DATA_BLOCK "Parameter"
{ S7_Optimized_Access := 'TRUE' }
VERSION : 0.1
NON_RETAIN
// ATTRIBUTES
// AUTO_NUMBER = False
// BLOCK_NUMBER = 170
// END_ATTRIBUTES
   VAR RETAIN
      AxisRun : Struct
         Axis { S7_SetPoint := 'False'} : Array[1..15] of "ServoType_UDT";
      END_STRUCT;
      AxisNuw : Struct
         Axis { S7_SetPoint := 'False'} : Array[1..15] of "ServoType_UDT";
      END_STRUCT;
      AxisDisplay : Struct
         Axis { S7_SetPoint := 'False'} : Array[1..15] of "ServoType_UDT";
      END_STRUCT;
      AxisSave : Struct
         Axis { S7_SetPoint := 'False'} : Array[1..15] of "ServoType_UDT";
      END_STRUCT;
      AxisStore : Array[1..15] of Struct
         Axis { S7_SetPoint := 'False'} : Array[1..15] of "ServoType_UDT";
      END_STRUCT;
   END_VAR


BEGIN
   AxisRun.Axis[1].Pos1.Position := 3.419;
   AxisRun.Axis[1].Pos1.Speed := 10000;
   AxisRun.Axis[1].Pos1.Reached := FALSE;
   AxisRun.Axis[1].Pos2.Position := 48.386;
   AxisRun.Axis[1].Pos2.Speed := 10000;
   AxisRun.Axis[1].Pos2.Reached := FALSE;
   AxisRun.Axis[1].Pos3.Position := 93.294;
   AxisRun.Axis[1].Pos3.Speed := 10000;
   AxisRun.Axis[1].Pos3.Reached := FALSE;
   AxisRun.Axis[1].Pos4.Position := 138.335;
   AxisRun.Axis[1].Pos4.Speed := 10000;
   AxisRun.Axis[1].Pos4.Reached := FALSE;
   AxisRun.Axis[1].Pos5.Position := 183.464;
   AxisRun.Axis[1].Pos5.Speed := 10000;
   AxisRun.Axis[1].Pos5.Reached := FALSE;
   AxisRun.Axis[1].Pos6.Position := 228.443;
   AxisRun.Axis[1].Pos6.Speed := 10000;
   AxisRun.Axis[1].Pos6.Reached := FALSE;
   AxisRun.Axis[1].Pos7.Position := 273.535;
   AxisRun.Axis[1].Pos7.Speed := 10000;
   AxisRun.Axis[1].Pos7.Reached := FALSE;
   AxisRun.Axis[1].Pos8.Position := 318.25;
   AxisRun.Axis[1].Pos8.Speed := 10000;
   AxisRun.Axis[1].Pos8.Reached := FALSE;
   AxisRun.Axis[1].Pos9.Position := 0.0;
   AxisRun.Axis[1].Pos9.Speed := 0;
   AxisRun.Axis[1].Pos9.Reached := FALSE;
   AxisRun.Axis[1].Pos10.Position := 0.0;
   AxisRun.Axis[1].Pos10.Speed := 0;
   AxisRun.Axis[1].Pos10.Reached := FALSE;
   AxisRun.Axis[1].Pos11.Position := 0.0;
   AxisRun.Axis[1].Pos11.Speed := 0;
   AxisRun.Axis[1].Pos11.Reached := FALSE;
   AxisRun.Axis[1].Pos12.Position := 0.0;
   AxisRun.Axis[1].Pos12.Speed := 0;
   AxisRun.Axis[1].Pos12.Reached := FALSE;
   AxisRun.Axis[1].Pos13.Position := 0.0;
   AxisRun.Axis[1].Pos13.Speed := 0;
   AxisRun.Axis[1].Pos13.Reached := FALSE;
   AxisRun.Axis[1].Pos14.Position := 0.0;
   AxisRun.Axis[1].Pos14.Speed := 0;
   AxisRun.Axis[1].Pos14.Reached := FALSE;
   AxisRun.Axis[1].Pos15.Position := 0.0;
   AxisRun.Axis[1].Pos15.Speed := 0;
   AxisRun.Axis[1].Pos15.Reached := FALSE;
   AxisRun.Axis[1].Pos16.Position := 0.0;
   AxisRun.Axis[1].Pos16.Speed := 0;
   AxisRun.Axis[1].Pos16.Reached := FALSE;
   AxisRun.Axis[1].Pos17.Position := 0.0;
   AxisRun.Axis[1].Pos17.Speed := 0;
   AxisRun.Axis[1].Pos17.Reached := FALSE;
   AxisRun.Axis[1].Pos18.Position := 0.0;
   AxisRun.Axis[1].Pos18.Speed := 0;
   AxisRun.Axis[1].Pos18.Reached := FALSE;
   AxisRun.Axis[1].Pos19.Position := 0.0;
   AxisRun.Axis[1].Pos19.Speed := 0;
   AxisRun.Axis[1].Pos19.Reached := FALSE;
   AxisRun.Axis[1].Pos20.Position := 0.0;
   AxisRun.Axis[1].Pos20.Speed := 0;
   AxisRun.Axis[1].Pos20.Reached := FALSE;
   AxisRun.Axis[1].Pos21.Position := 0.0;
   AxisRun.Axis[1].Pos21.Speed := 0;
   AxisRun.Axis[1].Pos21.Reached := FALSE;
   AxisRun.Axis[1].Pos22.Position := 0.0;
   AxisRun.Axis[1].Pos22.Speed := 0;
   AxisRun.Axis[1].Pos22.Reached := FALSE;
   AxisRun.Axis[1].Pos23.Position := 0.0;
   AxisRun.Axis[1].Pos23.Speed := 0;
   AxisRun.Axis[1].Pos23.Reached := FALSE;
   AxisRun.Axis[1].Pos24.Position := 0.0;
   AxisRun.Axis[1].Pos24.Speed := 0;
   AxisRun.Axis[1].Pos24.Reached := FALSE;
   AxisRun.Axis[1].Pos25.Position := 0.0;
   AxisRun.Axis[1].Pos25.Speed := 0;
   AxisRun.Axis[1].Pos25.Reached := FALSE;
   AxisRun.Axis[1].Pos26.Position := 0.0;
   AxisRun.Axis[1].Pos26.Speed := 0;
   AxisRun.Axis[1].Pos26.Reached := FALSE;
   AxisRun.Axis[1].Pos27.Position := 0.0;
   AxisRun.Axis[1].Pos27.Speed := 0;
   AxisRun.Axis[1].Pos27.Reached := FALSE;
   AxisRun.Axis[1].Pos28.Position := 0.0;
   AxisRun.Axis[1].Pos28.Speed := 0;
   AxisRun.Axis[1].Pos28.Reached := FALSE;
   AxisRun.Axis[1].Pos29.Position := 0.0;
   AxisRun.Axis[1].Pos29.Speed := 0;
   AxisRun.Axis[1].Pos29.Reached := FALSE;
   AxisRun.Axis[1].Pos30.Position := 0.0;
   AxisRun.Axis[1].Pos30.Speed := 0;
   AxisRun.Axis[1].Pos30.Reached := FALSE;
   AxisRun.Axis[2].Pos1.Position := 0.0;
   AxisRun.Axis[2].Pos1.Speed := 10000;
   AxisRun.Axis[2].Pos1.Reached := FALSE;
   AxisRun.Axis[2].Pos2.Position := 450.0;
   AxisRun.Axis[2].Pos2.Speed := 10000;
   AxisRun.Axis[2].Pos2.Reached := FALSE;
   AxisRun.Axis[2].Pos3.Position := 900.0;
   AxisRun.Axis[2].Pos3.Speed := 10000;
   AxisRun.Axis[2].Pos3.Reached := FALSE;
   AxisRun.Axis[2].Pos4.Position := 135.0;
   AxisRun.Axis[2].Pos4.Speed := 10000;
   AxisRun.Axis[2].Pos4.Reached := FALSE;
   AxisRun.Axis[2].Pos5.Position := 180.0;
   AxisRun.Axis[2].Pos5.Speed := 10000;
   AxisRun.Axis[2].Pos5.Reached := FALSE;
   AxisRun.Axis[2].Pos6.Position := 225.0;
   AxisRun.Axis[2].Pos6.Speed := 10000;
   AxisRun.Axis[2].Pos6.Reached := FALSE;
   AxisRun.Axis[2].Pos7.Position := 270.0;
   AxisRun.Axis[2].Pos7.Speed := 10000;
   AxisRun.Axis[2].Pos7.Reached := FALSE;
   AxisRun.Axis[2].Pos8.Position := 315.0;
   AxisRun.Axis[2].Pos8.Speed := 10000;
   AxisRun.Axis[2].Pos8.Reached := FALSE;
   AxisRun.Axis[2].Pos9.Position := 0.0;
   AxisRun.Axis[2].Pos9.Speed := 0;
   AxisRun.Axis[2].Pos9.Reached := FALSE;
   AxisRun.Axis[2].Pos10.Position := 0.0;
   AxisRun.Axis[2].Pos10.Speed := 0;
   AxisRun.Axis[2].Pos10.Reached := FALSE;
   AxisRun.Axis[2].Pos11.Position := 0.0;
   AxisRun.Axis[2].Pos11.Speed := 0;
   AxisRun.Axis[2].Pos11.Reached := FALSE;
   AxisRun.Axis[2].Pos12.Position := 0.0;
   AxisRun.Axis[2].Pos12.Speed := 0;
   AxisRun.Axis[2].Pos12.Reached := FALSE;
   AxisRun.Axis[2].Pos13.Position := 0.0;
   AxisRun.Axis[2].Pos13.Speed := 0;
   AxisRun.Axis[2].Pos13.Reached := FALSE;
   AxisRun.Axis[2].Pos14.Position := 0.0;
   AxisRun.Axis[2].Pos14.Speed := 0;
   AxisRun.Axis[2].Pos14.Reached := FALSE;
   AxisRun.Axis[2].Pos15.Position := 0.0;
   AxisRun.Axis[2].Pos15.Speed := 0;
   AxisRun.Axis[2].Pos15.Reached := FALSE;
   AxisRun.Axis[2].Pos16.Position := 0.0;
   AxisRun.Axis[2].Pos16.Speed := 0;
   AxisRun.Axis[2].Pos16.Reached := FALSE;
   AxisRun.Axis[2].Pos17.Position := 0.0;
   AxisRun.Axis[2].Pos17.Speed := 0;
   AxisRun.Axis[2].Pos17.Reached := FALSE;
   AxisRun.Axis[2].Pos18.Position := 0.0;
   AxisRun.Axis[2].Pos18.Speed := 0;
   AxisRun.Axis[2].Pos18.Reached := FALSE;
   AxisRun.Axis[2].Pos19.Position := 0.0;
   AxisRun.Axis[2].Pos19.Speed := 0;
   AxisRun.Axis[2].Pos19.Reached := FALSE;
   AxisRun.Axis[2].Pos20.Position := 0.0;
   AxisRun.Axis[2].Pos20.Speed := 0;
   AxisRun.Axis[2].Pos20.Reached := FALSE;
   AxisRun.Axis[2].Pos21.Position := 0.0;
   AxisRun.Axis[2].Pos21.Speed := 0;
   AxisRun.Axis[2].Pos21.Reached := FALSE;
   AxisRun.Axis[2].Pos22.Position := 0.0;
   AxisRun.Axis[2].Pos22.Speed := 0;
   AxisRun.Axis[2].Pos22.Reached := FALSE;
   AxisRun.Axis[2].Pos23.Position := 0.0;
   AxisRun.Axis[2].Pos23.Speed := 0;
   AxisRun.Axis[2].Pos23.Reached := FALSE;
   AxisRun.Axis[2].Pos24.Position := 0.0;
   AxisRun.Axis[2].Pos24.Speed := 0;
   AxisRun.Axis[2].Pos24.Reached := FALSE;
   AxisRun.Axis[2].Pos25.Position := 0.0;
   AxisRun.Axis[2].Pos25.Speed := 0;
   AxisRun.Axis[2].Pos25.Reached := FALSE;
   AxisRun.Axis[2].Pos26.Position := 0.0;
   AxisRun.Axis[2].Pos26.Speed := 0;
   AxisRun.Axis[2].Pos26.Reached := FALSE;
   AxisRun.Axis[2].Pos27.Position := 0.0;
   AxisRun.Axis[2].Pos27.Speed := 0;
   AxisRun.Axis[2].Pos27.Reached := FALSE;
   AxisRun.Axis[2].Pos28.Position := 0.0;
   AxisRun.Axis[2].Pos28.Speed := 0;
   AxisRun.Axis[2].Pos28.Reached := FALSE;
   AxisRun.Axis[2].Pos29.Position := 0.0;
   AxisRun.Axis[2].Pos29.Speed := 0;
   AxisRun.Axis[2].Pos29.Reached := FALSE;
   AxisRun.Axis[2].Pos30.Position := 0.0;
   AxisRun.Axis[2].Pos30.Speed := 0;
   AxisRun.Axis[2].Pos30.Reached := FALSE;
   AxisRun.Axis[3].Pos1.Position := 0.0;
   AxisRun.Axis[3].Pos1.Speed := 20000;
   AxisRun.Axis[3].Pos1.Reached := FALSE;
   AxisRun.Axis[3].Pos2.Position := 490.0;
   AxisRun.Axis[3].Pos2.Speed := 10000;
   AxisRun.Axis[3].Pos2.Reached := FALSE;
   AxisRun.Axis[3].Pos3.Position := 490.0;
   AxisRun.Axis[3].Pos3.Speed := 10000;
   AxisRun.Axis[3].Pos3.Reached := FALSE;
   AxisRun.Axis[3].Pos4.Position := 490.0;
   AxisRun.Axis[3].Pos4.Speed := 10000;
   AxisRun.Axis[3].Pos4.Reached := FALSE;
   AxisRun.Axis[3].Pos5.Position := 0.0;
   AxisRun.Axis[3].Pos5.Speed := 0;
   AxisRun.Axis[3].Pos5.Reached := FALSE;
   AxisRun.Axis[3].Pos6.Position := 490.0;
   AxisRun.Axis[3].Pos6.Speed := 10000;
   AxisRun.Axis[3].Pos6.Reached := FALSE;
   AxisRun.Axis[3].Pos7.Position := 90.0;
   AxisRun.Axis[3].Pos7.Speed := 10000;
   AxisRun.Axis[3].Pos7.Reached := FALSE;
   AxisRun.Axis[3].Pos8.Position := 180.0;
   AxisRun.Axis[3].Pos8.Speed := 10000;
   AxisRun.Axis[3].Pos8.Reached := FALSE;
   AxisRun.Axis[3].Pos9.Position := 270.0;
   AxisRun.Axis[3].Pos9.Speed := 10000;
   AxisRun.Axis[3].Pos9.Reached := FALSE;
   AxisRun.Axis[3].Pos10.Position := 0.0;
   AxisRun.Axis[3].Pos10.Speed := 0;
   AxisRun.Axis[3].Pos10.Reached := FALSE;
   AxisRun.Axis[3].Pos11.Position := 0.0;
   AxisRun.Axis[3].Pos11.Speed := 0;
   AxisRun.Axis[3].Pos11.Reached := FALSE;
   AxisRun.Axis[3].Pos12.Position := 0.0;
   AxisRun.Axis[3].Pos12.Speed := 0;
   AxisRun.Axis[3].Pos12.Reached := FALSE;
   AxisRun.Axis[3].Pos13.Position := 0.0;
   AxisRun.Axis[3].Pos13.Speed := 0;
   AxisRun.Axis[3].Pos13.Reached := FALSE;
   AxisRun.Axis[3].Pos14.Position := 0.0;
   AxisRun.Axis[3].Pos14.Speed := 0;
   AxisRun.Axis[3].Pos14.Reached := FALSE;
   AxisRun.Axis[3].Pos15.Position := 0.0;
   AxisRun.Axis[3].Pos15.Speed := 0;
   AxisRun.Axis[3].Pos15.Reached := FALSE;
   AxisRun.Axis[3].Pos16.Position := 0.0;
   AxisRun.Axis[3].Pos16.Speed := 0;
   AxisRun.Axis[3].Pos16.Reached := FALSE;
   AxisRun.Axis[3].Pos17.Position := 0.0;
   AxisRun.Axis[3].Pos17.Speed := 0;
   AxisRun.Axis[3].Pos17.Reached := FALSE;
   AxisRun.Axis[3].Pos18.Position := 0.0;
   AxisRun.Axis[3].Pos18.Speed := 0;
   AxisRun.Axis[3].Pos18.Reached := FALSE;
   AxisRun.Axis[3].Pos19.Position := 0.0;
   AxisRun.Axis[3].Pos19.Speed := 0;
   AxisRun.Axis[3].Pos19.Reached := FALSE;
   AxisRun.Axis[3].Pos20.Position := 0.0;
   AxisRun.Axis[3].Pos20.Speed := 0;
   AxisRun.Axis[3].Pos20.Reached := FALSE;
   AxisRun.Axis[3].Pos21.Position := 0.0;
   AxisRun.Axis[3].Pos21.Speed := 0;
   AxisRun.Axis[3].Pos21.Reached := FALSE;
   AxisRun.Axis[3].Pos22.Position := 0.0;
   AxisRun.Axis[3].Pos22.Speed := 0;
   AxisRun.Axis[3].Pos22.Reached := FALSE;
   AxisRun.Axis[3].Pos23.Position := 0.0;
   AxisRun.Axis[3].Pos23.Speed := 0;
   AxisRun.Axis[3].Pos23.Reached := FALSE;
   AxisRun.Axis[3].Pos24.Position := 0.0;
   AxisRun.Axis[3].Pos24.Speed := 0;
   AxisRun.Axis[3].Pos24.Reached := FALSE;
   AxisRun.Axis[3].Pos25.Position := 0.0;
   AxisRun.Axis[3].Pos25.Speed := 0;
   AxisRun.Axis[3].Pos25.Reached := FALSE;
   AxisRun.Axis[3].Pos26.Position := 0.0;
   AxisRun.Axis[3].Pos26.Speed := 0;
   AxisRun.Axis[3].Pos26.Reached := FALSE;
   AxisRun.Axis[3].Pos27.Position := 0.0;
   AxisRun.Axis[3].Pos27.Speed := 0;
   AxisRun.Axis[3].Pos27.Reached := FALSE;
   AxisRun.Axis[3].Pos28.Position := 0.0;
   AxisRun.Axis[3].Pos28.Speed := 0;
   AxisRun.Axis[3].Pos28.Reached := FALSE;
   AxisRun.Axis[3].Pos29.Position := 0.0;
   AxisRun.Axis[3].Pos29.Speed := 0;
   AxisRun.Axis[3].Pos29.Reached := FALSE;
   AxisRun.Axis[3].Pos30.Position := 0.0;
   AxisRun.Axis[3].Pos30.Speed := 0;
   AxisRun.Axis[3].Pos30.Reached := FALSE;
   AxisRun.Axis[4].Pos1.Position := 3.585;
   AxisRun.Axis[4].Pos1.Speed := 10000;
   AxisRun.Axis[4].Pos1.Reached := FALSE;
   AxisRun.Axis[4].Pos2.Position := 48.61;
   AxisRun.Axis[4].Pos2.Speed := 10000;
   AxisRun.Axis[4].Pos2.Reached := FALSE;
   AxisRun.Axis[4].Pos3.Position := 93.637;
   AxisRun.Axis[4].Pos3.Speed := 10000;
   AxisRun.Axis[4].Pos3.Reached := FALSE;
   AxisRun.Axis[4].Pos4.Position := 138.606;
   AxisRun.Axis[4].Pos4.Speed := 10000;
   AxisRun.Axis[4].Pos4.Reached := FALSE;
   AxisRun.Axis[4].Pos5.Position := 183.388;
   AxisRun.Axis[4].Pos5.Speed := 10000;
   AxisRun.Axis[4].Pos5.Reached := FALSE;
   AxisRun.Axis[4].Pos6.Position := 228.458;
   AxisRun.Axis[4].Pos6.Speed := 10000;
   AxisRun.Axis[4].Pos6.Reached := FALSE;
   AxisRun.Axis[4].Pos7.Position := 273.513;
   AxisRun.Axis[4].Pos7.Speed := 10000;
   AxisRun.Axis[4].Pos7.Reached := FALSE;
   AxisRun.Axis[4].Pos8.Position := 318.501;
   AxisRun.Axis[4].Pos8.Speed := 10000;
   AxisRun.Axis[4].Pos8.Reached := FALSE;
   AxisRun.Axis[4].Pos9.Position := 0.0;
   AxisRun.Axis[4].Pos9.Speed := 0;
   AxisRun.Axis[4].Pos9.Reached := FALSE;
   AxisRun.Axis[4].Pos10.Position := 0.0;
   AxisRun.Axis[4].Pos10.Speed := 0;
   AxisRun.Axis[4].Pos10.Reached := FALSE;
   AxisRun.Axis[4].Pos11.Position := 0.0;
   AxisRun.Axis[4].Pos11.Speed := 0;
   AxisRun.Axis[4].Pos11.Reached := FALSE;
   AxisRun.Axis[4].Pos12.Position := 0.0;
   AxisRun.Axis[4].Pos12.Speed := 0;
   AxisRun.Axis[4].Pos12.Reached := FALSE;
   AxisRun.Axis[4].Pos13.Position := 0.0;
   AxisRun.Axis[4].Pos13.Speed := 0;
   AxisRun.Axis[4].Pos13.Reached := FALSE;
   AxisRun.Axis[4].Pos14.Position := 0.0;
   AxisRun.Axis[4].Pos14.Speed := 0;
   AxisRun.Axis[4].Pos14.Reached := FALSE;
   AxisRun.Axis[4].Pos15.Position := 0.0;
   AxisRun.Axis[4].Pos15.Speed := 0;
   AxisRun.Axis[4].Pos15.Reached := FALSE;
   AxisRun.Axis[4].Pos16.Position := 0.0;
   AxisRun.Axis[4].Pos16.Speed := 0;
   AxisRun.Axis[4].Pos16.Reached := FALSE;
   AxisRun.Axis[4].Pos17.Position := 0.0;
   AxisRun.Axis[4].Pos17.Speed := 0;
   AxisRun.Axis[4].Pos17.Reached := FALSE;
   AxisRun.Axis[4].Pos18.Position := 0.0;
   AxisRun.Axis[4].Pos18.Speed := 0;
   AxisRun.Axis[4].Pos18.Reached := FALSE;
   AxisRun.Axis[4].Pos19.Position := 0.0;
   AxisRun.Axis[4].Pos19.Speed := 0;
   AxisRun.Axis[4].Pos19.Reached := FALSE;
   AxisRun.Axis[4].Pos20.Position := 0.0;
   AxisRun.Axis[4].Pos20.Speed := 0;
   AxisRun.Axis[4].Pos20.Reached := FALSE;
   AxisRun.Axis[4].Pos21.Position := 0.0;
   AxisRun.Axis[4].Pos21.Speed := 0;
   AxisRun.Axis[4].Pos21.Reached := FALSE;
   AxisRun.Axis[4].Pos22.Position := 0.0;
   AxisRun.Axis[4].Pos22.Speed := 0;
   AxisRun.Axis[4].Pos22.Reached := FALSE;
   AxisRun.Axis[4].Pos23.Position := 0.0;
   AxisRun.Axis[4].Pos23.Speed := 0;
   AxisRun.Axis[4].Pos23.Reached := FALSE;
   AxisRun.Axis[4].Pos24.Position := 0.0;
   AxisRun.Axis[4].Pos24.Speed := 0;
   AxisRun.Axis[4].Pos24.Reached := FALSE;
   AxisRun.Axis[4].Pos25.Position := 0.0;
   AxisRun.Axis[4].Pos25.Speed := 0;
   AxisRun.Axis[4].Pos25.Reached := FALSE;
   AxisRun.Axis[4].Pos26.Position := 0.0;
   AxisRun.Axis[4].Pos26.Speed := 0;
   AxisRun.Axis[4].Pos26.Reached := FALSE;
   AxisRun.Axis[4].Pos27.Position := 0.0;
   AxisRun.Axis[4].Pos27.Speed := 0;
   AxisRun.Axis[4].Pos27.Reached := FALSE;
   AxisRun.Axis[4].Pos28.Position := 0.0;
   AxisRun.Axis[4].Pos28.Speed := 0;
   AxisRun.Axis[4].Pos28.Reached := FALSE;
   AxisRun.Axis[4].Pos29.Position := 0.0;
   AxisRun.Axis[4].Pos29.Speed := 0;
   AxisRun.Axis[4].Pos29.Reached := FALSE;
   AxisRun.Axis[4].Pos30.Position := 0.0;
   AxisRun.Axis[4].Pos30.Speed := 0;
   AxisRun.Axis[4].Pos30.Reached := FALSE;
   AxisRun.Axis[5].Pos1.Position := 143.76;
   AxisRun.Axis[5].Pos1.Speed := 200;
   AxisRun.Axis[5].Pos1.Reached := FALSE;
   AxisRun.Axis[5].Pos2.Position := 143.76;
   AxisRun.Axis[5].Pos2.Speed := 200;
   AxisRun.Axis[5].Pos2.Reached := FALSE;
   AxisRun.Axis[5].Pos3.Position := 137.76;
   AxisRun.Axis[5].Pos3.Speed := 200;
   AxisRun.Axis[5].Pos3.Reached := FALSE;
   AxisRun.Axis[5].Pos4.Position := 130.36;
   AxisRun.Axis[5].Pos4.Speed := 200;
   AxisRun.Axis[5].Pos4.Reached := FALSE;
   AxisRun.Axis[5].Pos5.Position := 124.16;
   AxisRun.Axis[5].Pos5.Speed := 200;
   AxisRun.Axis[5].Pos5.Reached := FALSE;
   AxisRun.Axis[5].Pos6.Position := 125.65;
   AxisRun.Axis[5].Pos6.Speed := 200;
   AxisRun.Axis[5].Pos6.Reached := FALSE;
   AxisRun.Axis[5].Pos7.Position := 48.11;
   AxisRun.Axis[5].Pos7.Speed := 200;
   AxisRun.Axis[5].Pos7.Reached := FALSE;
   AxisRun.Axis[5].Pos8.Position := 0.0;
   AxisRun.Axis[5].Pos8.Speed := 200;
   AxisRun.Axis[5].Pos8.Reached := FALSE;
   AxisRun.Axis[5].Pos9.Position := 48.11;
   AxisRun.Axis[5].Pos9.Speed := 200;
   AxisRun.Axis[5].Pos9.Reached := FALSE;
   AxisRun.Axis[5].Pos10.Position := 0.0;
   AxisRun.Axis[5].Pos10.Speed := 0;
   AxisRun.Axis[5].Pos10.Reached := FALSE;
   AxisRun.Axis[5].Pos11.Position := 0.0;
   AxisRun.Axis[5].Pos11.Speed := 0;
   AxisRun.Axis[5].Pos11.Reached := FALSE;
   AxisRun.Axis[5].Pos12.Position := 0.0;
   AxisRun.Axis[5].Pos12.Speed := 0;
   AxisRun.Axis[5].Pos12.Reached := FALSE;
   AxisRun.Axis[5].Pos13.Position := 0.0;
   AxisRun.Axis[5].Pos13.Speed := 0;
   AxisRun.Axis[5].Pos13.Reached := FALSE;
   AxisRun.Axis[5].Pos14.Position := 0.0;
   AxisRun.Axis[5].Pos14.Speed := 0;
   AxisRun.Axis[5].Pos14.Reached := FALSE;
   AxisRun.Axis[5].Pos15.Position := 0.0;
   AxisRun.Axis[5].Pos15.Speed := 0;
   AxisRun.Axis[5].Pos15.Reached := FALSE;
   AxisRun.Axis[5].Pos16.Position := 0.0;
   AxisRun.Axis[5].Pos16.Speed := 0;
   AxisRun.Axis[5].Pos16.Reached := FALSE;
   AxisRun.Axis[5].Pos17.Position := 0.0;
   AxisRun.Axis[5].Pos17.Speed := 0;
   AxisRun.Axis[5].Pos17.Reached := FALSE;
   AxisRun.Axis[5].Pos18.Position := 0.0;
   AxisRun.Axis[5].Pos18.Speed := 0;
   AxisRun.Axis[5].Pos18.Reached := FALSE;
   AxisRun.Axis[5].Pos19.Position := 0.0;
   AxisRun.Axis[5].Pos19.Speed := 0;
   AxisRun.Axis[5].Pos19.Reached := FALSE;
   AxisRun.Axis[5].Pos20.Position := 0.0;
   AxisRun.Axis[5].Pos20.Speed := 0;
   AxisRun.Axis[5].Pos20.Reached := FALSE;
   AxisRun.Axis[5].Pos21.Position := 0.0;
   AxisRun.Axis[5].Pos21.Speed := 0;
   AxisRun.Axis[5].Pos21.Reached := FALSE;
   AxisRun.Axis[5].Pos22.Position := 0.0;
   AxisRun.Axis[5].Pos22.Speed := 0;
   AxisRun.Axis[5].Pos22.Reached := FALSE;
   AxisRun.Axis[5].Pos23.Position := 0.0;
   AxisRun.Axis[5].Pos23.Speed := 0;
   AxisRun.Axis[5].Pos23.Reached := FALSE;
   AxisRun.Axis[5].Pos24.Position := 0.0;
   AxisRun.Axis[5].Pos24.Speed := 0;
   AxisRun.Axis[5].Pos24.Reached := FALSE;
   AxisRun.Axis[5].Pos25.Position := 0.0;
   AxisRun.Axis[5].Pos25.Speed := 0;
   AxisRun.Axis[5].Pos25.Reached := FALSE;
   AxisRun.Axis[5].Pos26.Position := 0.0;
   AxisRun.Axis[5].Pos26.Speed := 0;
   AxisRun.Axis[5].Pos26.Reached := FALSE;
   AxisRun.Axis[5].Pos27.Position := 0.0;
   AxisRun.Axis[5].Pos27.Speed := 0;
   AxisRun.Axis[5].Pos27.Reached := FALSE;
   AxisRun.Axis[5].Pos28.Position := 0.0;
   AxisRun.Axis[5].Pos28.Speed := 0;
   AxisRun.Axis[5].Pos28.Reached := FALSE;
   AxisRun.Axis[5].Pos29.Position := 0.0;
   AxisRun.Axis[5].Pos29.Speed := 0;
   AxisRun.Axis[5].Pos29.Reached := FALSE;
   AxisRun.Axis[5].Pos30.Position := 0.0;
   AxisRun.Axis[5].Pos30.Speed := 0;
   AxisRun.Axis[5].Pos30.Reached := FALSE;
   AxisRun.Axis[6].Pos1.Position := 2.34;
   AxisRun.Axis[6].Pos1.Speed := 200;
   AxisRun.Axis[6].Pos1.Reached := FALSE;
   AxisRun.Axis[6].Pos2.Position := 76.0;
   AxisRun.Axis[6].Pos2.Speed := 200;
   AxisRun.Axis[6].Pos2.Reached := FALSE;
   AxisRun.Axis[6].Pos3.Position := 84.69;
   AxisRun.Axis[6].Pos3.Speed := 200;
   AxisRun.Axis[6].Pos3.Reached := FALSE;
   AxisRun.Axis[6].Pos4.Position := 84.69;
   AxisRun.Axis[6].Pos4.Speed := 200;
   AxisRun.Axis[6].Pos4.Reached := FALSE;
   AxisRun.Axis[6].Pos5.Position := 84.69;
   AxisRun.Axis[6].Pos5.Speed := 200;
   AxisRun.Axis[6].Pos5.Reached := FALSE;
   AxisRun.Axis[6].Pos6.Position := 84.69;
   AxisRun.Axis[6].Pos6.Speed := 200;
   AxisRun.Axis[6].Pos6.Reached := FALSE;
   AxisRun.Axis[6].Pos7.Position := 85.0;
   AxisRun.Axis[6].Pos7.Speed := 200;
   AxisRun.Axis[6].Pos7.Reached := FALSE;
   AxisRun.Axis[6].Pos8.Position := 88.53;
   AxisRun.Axis[6].Pos8.Speed := 200;
   AxisRun.Axis[6].Pos8.Reached := FALSE;
   AxisRun.Axis[6].Pos9.Position := 0.0;
   AxisRun.Axis[6].Pos9.Speed := 0;
   AxisRun.Axis[6].Pos9.Reached := FALSE;
   AxisRun.Axis[6].Pos10.Position := 0.0;
   AxisRun.Axis[6].Pos10.Speed := 0;
   AxisRun.Axis[6].Pos10.Reached := FALSE;
   AxisRun.Axis[6].Pos11.Position := 0.0;
   AxisRun.Axis[6].Pos11.Speed := 0;
   AxisRun.Axis[6].Pos11.Reached := FALSE;
   AxisRun.Axis[6].Pos12.Position := 0.0;
   AxisRun.Axis[6].Pos12.Speed := 0;
   AxisRun.Axis[6].Pos12.Reached := FALSE;
   AxisRun.Axis[6].Pos13.Position := 0.0;
   AxisRun.Axis[6].Pos13.Speed := 0;
   AxisRun.Axis[6].Pos13.Reached := FALSE;
   AxisRun.Axis[6].Pos14.Position := 0.0;
   AxisRun.Axis[6].Pos14.Speed := 0;
   AxisRun.Axis[6].Pos14.Reached := FALSE;
   AxisRun.Axis[6].Pos15.Position := 0.0;
   AxisRun.Axis[6].Pos15.Speed := 0;
   AxisRun.Axis[6].Pos15.Reached := FALSE;
   AxisRun.Axis[6].Pos16.Position := 0.0;
   AxisRun.Axis[6].Pos16.Speed := 0;
   AxisRun.Axis[6].Pos16.Reached := FALSE;
   AxisRun.Axis[6].Pos17.Position := 0.0;
   AxisRun.Axis[6].Pos17.Speed := 0;
   AxisRun.Axis[6].Pos17.Reached := FALSE;
   AxisRun.Axis[6].Pos18.Position := 0.0;
   AxisRun.Axis[6].Pos18.Speed := 0;
   AxisRun.Axis[6].Pos18.Reached := FALSE;
   AxisRun.Axis[6].Pos19.Position := 0.0;
   AxisRun.Axis[6].Pos19.Speed := 0;
   AxisRun.Axis[6].Pos19.Reached := FALSE;
   AxisRun.Axis[6].Pos20.Position := 0.0;
   AxisRun.Axis[6].Pos20.Speed := 0;
   AxisRun.Axis[6].Pos20.Reached := FALSE;
   AxisRun.Axis[6].Pos21.Position := 0.0;
   AxisRun.Axis[6].Pos21.Speed := 0;
   AxisRun.Axis[6].Pos21.Reached := FALSE;
   AxisRun.Axis[6].Pos22.Position := 0.0;
   AxisRun.Axis[6].Pos22.Speed := 0;
   AxisRun.Axis[6].Pos22.Reached := FALSE;
   AxisRun.Axis[6].Pos23.Position := 0.0;
   AxisRun.Axis[6].Pos23.Speed := 0;
   AxisRun.Axis[6].Pos23.Reached := FALSE;
   AxisRun.Axis[6].Pos24.Position := 0.0;
   AxisRun.Axis[6].Pos24.Speed := 0;
   AxisRun.Axis[6].Pos24.Reached := FALSE;
   AxisRun.Axis[6].Pos25.Position := 0.0;
   AxisRun.Axis[6].Pos25.Speed := 0;
   AxisRun.Axis[6].Pos25.Reached := FALSE;
   AxisRun.Axis[6].Pos26.Position := 0.0;
   AxisRun.Axis[6].Pos26.Speed := 0;
   AxisRun.Axis[6].Pos26.Reached := FALSE;
   AxisRun.Axis[6].Pos27.Position := 0.0;
   AxisRun.Axis[6].Pos27.Speed := 0;
   AxisRun.Axis[6].Pos27.Reached := FALSE;
   AxisRun.Axis[6].Pos28.Position := 0.0;
   AxisRun.Axis[6].Pos28.Speed := 0;
   AxisRun.Axis[6].Pos28.Reached := FALSE;
   AxisRun.Axis[6].Pos29.Position := 0.0;
   AxisRun.Axis[6].Pos29.Speed := 0;
   AxisRun.Axis[6].Pos29.Reached := FALSE;
   AxisRun.Axis[6].Pos30.Position := 0.0;
   AxisRun.Axis[6].Pos30.Speed := 0;
   AxisRun.Axis[6].Pos30.Reached := FALSE;
   AxisRun.Axis[7].Pos1.Position := 115.47;
   AxisRun.Axis[7].Pos1.Speed := 200;
   AxisRun.Axis[7].Pos1.Reached := FALSE;
   AxisRun.Axis[7].Pos2.Position := 115.47;
   AxisRun.Axis[7].Pos2.Speed := 200;
   AxisRun.Axis[7].Pos2.Reached := FALSE;
   AxisRun.Axis[7].Pos3.Position := 115.47;
   AxisRun.Axis[7].Pos3.Speed := 200;
   AxisRun.Axis[7].Pos3.Reached := FALSE;
   AxisRun.Axis[7].Pos4.Position := 115.47;
   AxisRun.Axis[7].Pos4.Speed := 200;
   AxisRun.Axis[7].Pos4.Reached := FALSE;
   AxisRun.Axis[7].Pos5.Position := 115.47;
   AxisRun.Axis[7].Pos5.Speed := 200;
   AxisRun.Axis[7].Pos5.Reached := FALSE;
   AxisRun.Axis[7].Pos6.Position := 110.18;
   AxisRun.Axis[7].Pos6.Speed := 200;
   AxisRun.Axis[7].Pos6.Reached := FALSE;
   AxisRun.Axis[7].Pos7.Position := 60.52;
   AxisRun.Axis[7].Pos7.Speed := 200;
   AxisRun.Axis[7].Pos7.Reached := FALSE;
   AxisRun.Axis[7].Pos8.Position := 80.0;
   AxisRun.Axis[7].Pos8.Speed := 100;
   AxisRun.Axis[7].Pos8.Reached := FALSE;
   AxisRun.Axis[7].Pos9.Position := 0.0;
   AxisRun.Axis[7].Pos9.Speed := 0;
   AxisRun.Axis[7].Pos9.Reached := FALSE;
   AxisRun.Axis[7].Pos10.Position := 0.0;
   AxisRun.Axis[7].Pos10.Speed := 0;
   AxisRun.Axis[7].Pos10.Reached := FALSE;
   AxisRun.Axis[7].Pos11.Position := 0.0;
   AxisRun.Axis[7].Pos11.Speed := 0;
   AxisRun.Axis[7].Pos11.Reached := FALSE;
   AxisRun.Axis[7].Pos12.Position := 0.0;
   AxisRun.Axis[7].Pos12.Speed := 0;
   AxisRun.Axis[7].Pos12.Reached := FALSE;
   AxisRun.Axis[7].Pos13.Position := 0.0;
   AxisRun.Axis[7].Pos13.Speed := 0;
   AxisRun.Axis[7].Pos13.Reached := FALSE;
   AxisRun.Axis[7].Pos14.Position := 0.0;
   AxisRun.Axis[7].Pos14.Speed := 0;
   AxisRun.Axis[7].Pos14.Reached := FALSE;
   AxisRun.Axis[7].Pos15.Position := 0.0;
   AxisRun.Axis[7].Pos15.Speed := 0;
   AxisRun.Axis[7].Pos15.Reached := FALSE;
   AxisRun.Axis[7].Pos16.Position := 0.0;
   AxisRun.Axis[7].Pos16.Speed := 0;
   AxisRun.Axis[7].Pos16.Reached := FALSE;
   AxisRun.Axis[7].Pos17.Position := 0.0;
   AxisRun.Axis[7].Pos17.Speed := 0;
   AxisRun.Axis[7].Pos17.Reached := FALSE;
   AxisRun.Axis[7].Pos18.Position := 0.0;
   AxisRun.Axis[7].Pos18.Speed := 0;
   AxisRun.Axis[7].Pos18.Reached := FALSE;
   AxisRun.Axis[7].Pos19.Position := 0.0;
   AxisRun.Axis[7].Pos19.Speed := 0;
   AxisRun.Axis[7].Pos19.Reached := FALSE;
   AxisRun.Axis[7].Pos20.Position := 0.0;
   AxisRun.Axis[7].Pos20.Speed := 0;
   AxisRun.Axis[7].Pos20.Reached := FALSE;
   AxisRun.Axis[7].Pos21.Position := 0.0;
   AxisRun.Axis[7].Pos21.Speed := 0;
   AxisRun.Axis[7].Pos21.Reached := FALSE;
   AxisRun.Axis[7].Pos22.Position := 0.0;
   AxisRun.Axis[7].Pos22.Speed := 0;
   AxisRun.Axis[7].Pos22.Reached := FALSE;
   AxisRun.Axis[7].Pos23.Position := 0.0;
   AxisRun.Axis[7].Pos23.Speed := 0;
   AxisRun.Axis[7].Pos23.Reached := FALSE;
   AxisRun.Axis[7].Pos24.Position := 0.0;
   AxisRun.Axis[7].Pos24.Speed := 0;
   AxisRun.Axis[7].Pos24.Reached := FALSE;
   AxisRun.Axis[7].Pos25.Position := 0.0;
   AxisRun.Axis[7].Pos25.Speed := 0;
   AxisRun.Axis[7].Pos25.Reached := FALSE;
   AxisRun.Axis[7].Pos26.Position := 0.0;
   AxisRun.Axis[7].Pos26.Speed := 0;
   AxisRun.Axis[7].Pos26.Reached := FALSE;
   AxisRun.Axis[7].Pos27.Position := 0.0;
   AxisRun.Axis[7].Pos27.Speed := 0;
   AxisRun.Axis[7].Pos27.Reached := FALSE;
   AxisRun.Axis[7].Pos28.Position := 0.0;
   AxisRun.Axis[7].Pos28.Speed := 0;
   AxisRun.Axis[7].Pos28.Reached := FALSE;
   AxisRun.Axis[7].Pos29.Position := 0.0;
   AxisRun.Axis[7].Pos29.Speed := 0;
   AxisRun.Axis[7].Pos29.Reached := FALSE;
   AxisRun.Axis[7].Pos30.Position := 0.0;
   AxisRun.Axis[7].Pos30.Speed := 0;
   AxisRun.Axis[7].Pos30.Reached := FALSE;
   AxisRun.Axis[8].Pos1.Position := 0.0;
   AxisRun.Axis[8].Pos1.Speed := 0;
   AxisRun.Axis[8].Pos1.Reached := FALSE;
   AxisRun.Axis[8].Pos2.Position := 0.0;
   AxisRun.Axis[8].Pos2.Speed := 0;
   AxisRun.Axis[8].Pos2.Reached := FALSE;
   AxisRun.Axis[8].Pos3.Position := 0.0;
   AxisRun.Axis[8].Pos3.Speed := 0;
   AxisRun.Axis[8].Pos3.Reached := FALSE;
   AxisRun.Axis[8].Pos4.Position := 0.0;
   AxisRun.Axis[8].Pos4.Speed := 0;
   AxisRun.Axis[8].Pos4.Reached := FALSE;
   AxisRun.Axis[8].Pos5.Position := 0.0;
   AxisRun.Axis[8].Pos5.Speed := 0;
   AxisRun.Axis[8].Pos5.Reached := FALSE;
   AxisRun.Axis[8].Pos6.Position := 0.0;
   AxisRun.Axis[8].Pos6.Speed := 0;
   AxisRun.Axis[8].Pos6.Reached := FALSE;
   AxisRun.Axis[8].Pos7.Position := 0.0;
   AxisRun.Axis[8].Pos7.Speed := 0;
   AxisRun.Axis[8].Pos7.Reached := FALSE;
   AxisRun.Axis[8].Pos8.Position := 0.0;
   AxisRun.Axis[8].Pos8.Speed := 0;
   AxisRun.Axis[8].Pos8.Reached := FALSE;
   AxisRun.Axis[8].Pos9.Position := 0.0;
   AxisRun.Axis[8].Pos9.Speed := 0;
   AxisRun.Axis[8].Pos9.Reached := FALSE;
   AxisRun.Axis[8].Pos10.Position := 0.0;
   AxisRun.Axis[8].Pos10.Speed := 0;
   AxisRun.Axis[8].Pos10.Reached := FALSE;
   AxisRun.Axis[8].Pos11.Position := 0.0;
   AxisRun.Axis[8].Pos11.Speed := 0;
   AxisRun.Axis[8].Pos11.Reached := FALSE;
   AxisRun.Axis[8].Pos12.Position := 0.0;
   AxisRun.Axis[8].Pos12.Speed := 0;
   AxisRun.Axis[8].Pos12.Reached := FALSE;
   AxisRun.Axis[8].Pos13.Position := 0.0;
   AxisRun.Axis[8].Pos13.Speed := 0;
   AxisRun.Axis[8].Pos13.Reached := FALSE;
   AxisRun.Axis[8].Pos14.Position := 0.0;
   AxisRun.Axis[8].Pos14.Speed := 0;
   AxisRun.Axis[8].Pos14.Reached := FALSE;
   AxisRun.Axis[8].Pos15.Position := 0.0;
   AxisRun.Axis[8].Pos15.Speed := 0;
   AxisRun.Axis[8].Pos15.Reached := FALSE;
   AxisRun.Axis[8].Pos16.Position := 0.0;
   AxisRun.Axis[8].Pos16.Speed := 0;
   AxisRun.Axis[8].Pos16.Reached := FALSE;
   AxisRun.Axis[8].Pos17.Position := 0.0;
   AxisRun.Axis[8].Pos17.Speed := 0;
   AxisRun.Axis[8].Pos17.Reached := FALSE;
   AxisRun.Axis[8].Pos18.Position := 0.0;
   AxisRun.Axis[8].Pos18.Speed := 0;
   AxisRun.Axis[8].Pos18.Reached := FALSE;
   AxisRun.Axis[8].Pos19.Position := 0.0;
   AxisRun.Axis[8].Pos19.Speed := 0;
   AxisRun.Axis[8].Pos19.Reached := FALSE;
   AxisRun.Axis[8].Pos20.Position := 0.0;
   AxisRun.Axis[8].Pos20.Speed := 0;
   AxisRun.Axis[8].Pos20.Reached := FALSE;
   AxisRun.Axis[8].Pos21.Position := 0.0;
   AxisRun.Axis[8].Pos21.Speed := 0;
   AxisRun.Axis[8].Pos21.Reached := FALSE;
   AxisRun.Axis[8].Pos22.Position := 0.0;
   AxisRun.Axis[8].Pos22.Speed := 0;
   AxisRun.Axis[8].Pos22.Reached := FALSE;
   AxisRun.Axis[8].Pos23.Position := 0.0;
   AxisRun.Axis[8].Pos23.Speed := 0;
   AxisRun.Axis[8].Pos23.Reached := FALSE;
   AxisRun.Axis[8].Pos24.Position := 0.0;
   AxisRun.Axis[8].Pos24.Speed := 0;
   AxisRun.Axis[8].Pos24.Reached := FALSE;
   AxisRun.Axis[8].Pos25.Position := 0.0;
   AxisRun.Axis[8].Pos25.Speed := 0;
   AxisRun.Axis[8].Pos25.Reached := FALSE;
   AxisRun.Axis[8].Pos26.Position := 0.0;
   AxisRun.Axis[8].Pos26.Speed := 0;
   AxisRun.Axis[8].Pos26.Reached := FALSE;
   AxisRun.Axis[8].Pos27.Position := 0.0;
   AxisRun.Axis[8].Pos27.Speed := 0;
   AxisRun.Axis[8].Pos27.Reached := FALSE;
   AxisRun.Axis[8].Pos28.Position := 0.0;
   AxisRun.Axis[8].Pos28.Speed := 0;
   AxisRun.Axis[8].Pos28.Reached := FALSE;
   AxisRun.Axis[8].Pos29.Position := 0.0;
   AxisRun.Axis[8].Pos29.Speed := 0;
   AxisRun.Axis[8].Pos29.Reached := FALSE;
   AxisRun.Axis[8].Pos30.Position := 0.0;
   AxisRun.Axis[8].Pos30.Speed := 0;
   AxisRun.Axis[8].Pos30.Reached := FALSE;
   AxisRun.Axis[9].Pos1.Position := 0.0;
   AxisRun.Axis[9].Pos1.Speed := 0;
   AxisRun.Axis[9].Pos1.Reached := FALSE;
   AxisRun.Axis[9].Pos2.Position := 0.0;
   AxisRun.Axis[9].Pos2.Speed := 0;
   AxisRun.Axis[9].Pos2.Reached := FALSE;
   AxisRun.Axis[9].Pos3.Position := 0.0;
   AxisRun.Axis[9].Pos3.Speed := 0;
   AxisRun.Axis[9].Pos3.Reached := FALSE;
   AxisRun.Axis[9].Pos4.Position := 0.0;
   AxisRun.Axis[9].Pos4.Speed := 0;
   AxisRun.Axis[9].Pos4.Reached := FALSE;
   AxisRun.Axis[9].Pos5.Position := 0.0;
   AxisRun.Axis[9].Pos5.Speed := 0;
   AxisRun.Axis[9].Pos5.Reached := FALSE;
   AxisRun.Axis[9].Pos6.Position := 0.0;
   AxisRun.Axis[9].Pos6.Speed := 0;
   AxisRun.Axis[9].Pos6.Reached := FALSE;
   AxisRun.Axis[9].Pos7.Position := 0.0;
   AxisRun.Axis[9].Pos7.Speed := 0;
   AxisRun.Axis[9].Pos7.Reached := FALSE;
   AxisRun.Axis[9].Pos8.Position := 0.0;
   AxisRun.Axis[9].Pos8.Speed := 0;
   AxisRun.Axis[9].Pos8.Reached := FALSE;
   AxisRun.Axis[9].Pos9.Position := 0.0;
   AxisRun.Axis[9].Pos9.Speed := 0;
   AxisRun.Axis[9].Pos9.Reached := FALSE;
   AxisRun.Axis[9].Pos10.Position := 0.0;
   AxisRun.Axis[9].Pos10.Speed := 0;
   AxisRun.Axis[9].Pos10.Reached := FALSE;
   AxisRun.Axis[9].Pos11.Position := 0.0;
   AxisRun.Axis[9].Pos11.Speed := 0;
   AxisRun.Axis[9].Pos11.Reached := FALSE;
   AxisRun.Axis[9].Pos12.Position := 0.0;
   AxisRun.Axis[9].Pos12.Speed := 0;
   AxisRun.Axis[9].Pos12.Reached := FALSE;
   AxisRun.Axis[9].Pos13.Position := 0.0;
   AxisRun.Axis[9].Pos13.Speed := 0;
   AxisRun.Axis[9].Pos13.Reached := FALSE;
   AxisRun.Axis[9].Pos14.Position := 0.0;
   AxisRun.Axis[9].Pos14.Speed := 0;
   AxisRun.Axis[9].Pos14.Reached := FALSE;
   AxisRun.Axis[9].Pos15.Position := 0.0;
   AxisRun.Axis[9].Pos15.Speed := 0;
   AxisRun.Axis[9].Pos15.Reached := FALSE;
   AxisRun.Axis[9].Pos16.Position := 0.0;
   AxisRun.Axis[9].Pos16.Speed := 0;
   AxisRun.Axis[9].Pos16.Reached := FALSE;
   AxisRun.Axis[9].Pos17.Position := 0.0;
   AxisRun.Axis[9].Pos17.Speed := 0;
   AxisRun.Axis[9].Pos17.Reached := FALSE;
   AxisRun.Axis[9].Pos18.Position := 0.0;
   AxisRun.Axis[9].Pos18.Speed := 0;
   AxisRun.Axis[9].Pos18.Reached := FALSE;
   AxisRun.Axis[9].Pos19.Position := 0.0;
   AxisRun.Axis[9].Pos19.Speed := 0;
   AxisRun.Axis[9].Pos19.Reached := FALSE;
   AxisRun.Axis[9].Pos20.Position := 0.0;
   AxisRun.Axis[9].Pos20.Speed := 0;
   AxisRun.Axis[9].Pos20.Reached := FALSE;
   AxisRun.Axis[9].Pos21.Position := 0.0;
   AxisRun.Axis[9].Pos21.Speed := 0;
   AxisRun.Axis[9].Pos21.Reached := FALSE;
   AxisRun.Axis[9].Pos22.Position := 0.0;
   AxisRun.Axis[9].Pos22.Speed := 0;
   AxisRun.Axis[9].Pos22.Reached := FALSE;
   AxisRun.Axis[9].Pos23.Position := 0.0;
   AxisRun.Axis[9].Pos23.Speed := 0;
   AxisRun.Axis[9].Pos23.Reached := FALSE;
   AxisRun.Axis[9].Pos24.Position := 0.0;
   AxisRun.Axis[9].Pos24.Speed := 0;
   AxisRun.Axis[9].Pos24.Reached := FALSE;
   AxisRun.Axis[9].Pos25.Position := 0.0;
   AxisRun.Axis[9].Pos25.Speed := 0;
   AxisRun.Axis[9].Pos25.Reached := FALSE;
   AxisRun.Axis[9].Pos26.Position := 0.0;
   AxisRun.Axis[9].Pos26.Speed := 0;
   AxisRun.Axis[9].Pos26.Reached := FALSE;
   AxisRun.Axis[9].Pos27.Position := 0.0;
   AxisRun.Axis[9].Pos27.Speed := 0;
   AxisRun.Axis[9].Pos27.Reached := FALSE;
   AxisRun.Axis[9].Pos28.Position := 0.0;
   AxisRun.Axis[9].Pos28.Speed := 0;
   AxisRun.Axis[9].Pos28.Reached := FALSE;
   AxisRun.Axis[9].Pos29.Position := 0.0;
   AxisRun.Axis[9].Pos29.Speed := 0;
   AxisRun.Axis[9].Pos29.Reached := FALSE;
   AxisRun.Axis[9].Pos30.Position := 0.0;
   AxisRun.Axis[9].Pos30.Speed := 0;
   AxisRun.Axis[9].Pos30.Reached := FALSE;
   AxisRun.Axis[10].Pos1.Position := 0.0;
   AxisRun.Axis[10].Pos1.Speed := 0;
   AxisRun.Axis[10].Pos1.Reached := FALSE;
   AxisRun.Axis[10].Pos2.Position := 0.0;
   AxisRun.Axis[10].Pos2.Speed := 0;
   AxisRun.Axis[10].Pos2.Reached := FALSE;
   AxisRun.Axis[10].Pos3.Position := 0.0;
   AxisRun.Axis[10].Pos3.Speed := 0;
   AxisRun.Axis[10].Pos3.Reached := FALSE;
   AxisRun.Axis[10].Pos4.Position := 0.0;
   AxisRun.Axis[10].Pos4.Speed := 0;
   AxisRun.Axis[10].Pos4.Reached := FALSE;
   AxisRun.Axis[10].Pos5.Position := 0.0;
   AxisRun.Axis[10].Pos5.Speed := 0;
   AxisRun.Axis[10].Pos5.Reached := FALSE;
   AxisRun.Axis[10].Pos6.Position := 0.0;
   AxisRun.Axis[10].Pos6.Speed := 0;
   AxisRun.Axis[10].Pos6.Reached := FALSE;
   AxisRun.Axis[10].Pos7.Position := 0.0;
   AxisRun.Axis[10].Pos7.Speed := 0;
   AxisRun.Axis[10].Pos7.Reached := FALSE;
   AxisRun.Axis[10].Pos8.Position := 0.0;
   AxisRun.Axis[10].Pos8.Speed := 0;
   AxisRun.Axis[10].Pos8.Reached := FALSE;
   AxisRun.Axis[10].Pos9.Position := 0.0;
   AxisRun.Axis[10].Pos9.Speed := 0;
   AxisRun.Axis[10].Pos9.Reached := FALSE;
   AxisRun.Axis[10].Pos10.Position := 0.0;
   AxisRun.Axis[10].Pos10.Speed := 0;
   AxisRun.Axis[10].Pos10.Reached := FALSE;
   AxisRun.Axis[10].Pos11.Position := 0.0;
   AxisRun.Axis[10].Pos11.Speed := 0;
   AxisRun.Axis[10].Pos11.Reached := FALSE;
   AxisRun.Axis[10].Pos12.Position := 0.0;
   AxisRun.Axis[10].Pos12.Speed := 0;
   AxisRun.Axis[10].Pos12.Reached := FALSE;
   AxisRun.Axis[10].Pos13.Position := 0.0;
   AxisRun.Axis[10].Pos13.Speed := 0;
   AxisRun.Axis[10].Pos13.Reached := FALSE;
   AxisRun.Axis[10].Pos14.Position := 0.0;
   AxisRun.Axis[10].Pos14.Speed := 0;
   AxisRun.Axis[10].Pos14.Reached := FALSE;
   AxisRun.Axis[10].Pos15.Position := 0.0;
   AxisRun.Axis[10].Pos15.Speed := 0;
   AxisRun.Axis[10].Pos15.Reached := FALSE;
   AxisRun.Axis[10].Pos16.Position := 0.0;
   AxisRun.Axis[10].Pos16.Speed := 0;
   AxisRun.Axis[10].Pos16.Reached := FALSE;
   AxisRun.Axis[10].Pos17.Position := 0.0;
   AxisRun.Axis[10].Pos17.Speed := 0;
   AxisRun.Axis[10].Pos17.Reached := FALSE;
   AxisRun.Axis[10].Pos18.Position := 0.0;
   AxisRun.Axis[10].Pos18.Speed := 0;
   AxisRun.Axis[10].Pos18.Reached := FALSE;
   AxisRun.Axis[10].Pos19.Position := 0.0;
   AxisRun.Axis[10].Pos19.Speed := 0;
   AxisRun.Axis[10].Pos19.Reached := FALSE;
   AxisRun.Axis[10].Pos20.Position := 0.0;
   AxisRun.Axis[10].Pos20.Speed := 0;
   AxisRun.Axis[10].Pos20.Reached := FALSE;
   AxisRun.Axis[10].Pos21.Position := 0.0;
   AxisRun.Axis[10].Pos21.Speed := 0;
   AxisRun.Axis[10].Pos21.Reached := FALSE;
   AxisRun.Axis[10].Pos22.Position := 0.0;
   AxisRun.Axis[10].Pos22.Speed := 0;
   AxisRun.Axis[10].Pos22.Reached := FALSE;
   AxisRun.Axis[10].Pos23.Position := 0.0;
   AxisRun.Axis[10].Pos23.Speed := 0;
   AxisRun.Axis[10].Pos23.Reached := FALSE;
   AxisRun.Axis[10].Pos24.Position := 0.0;
   AxisRun.Axis[10].Pos24.Speed := 0;
   AxisRun.Axis[10].Pos24.Reached := FALSE;
   AxisRun.Axis[10].Pos25.Position := 0.0;
   AxisRun.Axis[10].Pos25.Speed := 0;
   AxisRun.Axis[10].Pos25.Reached := FALSE;
   AxisRun.Axis[10].Pos26.Position := 0.0;
   AxisRun.Axis[10].Pos26.Speed := 0;
   AxisRun.Axis[10].Pos26.Reached := FALSE;
   AxisRun.Axis[10].Pos27.Position := 0.0;
   AxisRun.Axis[10].Pos27.Speed := 0;
   AxisRun.Axis[10].Pos27.Reached := FALSE;
   AxisRun.Axis[10].Pos28.Position := 0.0;
   AxisRun.Axis[10].Pos28.Speed := 0;
   AxisRun.Axis[10].Pos28.Reached := FALSE;
   AxisRun.Axis[10].Pos29.Position := 0.0;
   AxisRun.Axis[10].Pos29.Speed := 0;
   AxisRun.Axis[10].Pos29.Reached := FALSE;
   AxisRun.Axis[10].Pos30.Position := 0.0;
   AxisRun.Axis[10].Pos30.Speed := 0;
   AxisRun.Axis[10].Pos30.Reached := FALSE;
   AxisRun.Axis[11].Pos1.Position := 0.0;
   AxisRun.Axis[11].Pos1.Speed := 0;
   AxisRun.Axis[11].Pos1.Reached := FALSE;
   AxisRun.Axis[11].Pos2.Position := 0.0;
   AxisRun.Axis[11].Pos2.Speed := 0;
   AxisRun.Axis[11].Pos2.Reached := FALSE;
   AxisRun.Axis[11].Pos3.Position := 0.0;
   AxisRun.Axis[11].Pos3.Speed := 0;
   AxisRun.Axis[11].Pos3.Reached := FALSE;
   AxisRun.Axis[11].Pos4.Position := 0.0;
   AxisRun.Axis[11].Pos4.Speed := 0;
   AxisRun.Axis[11].Pos4.Reached := FALSE;
   AxisRun.Axis[11].Pos5.Position := 0.0;
   AxisRun.Axis[11].Pos5.Speed := 0;
   AxisRun.Axis[11].Pos5.Reached := FALSE;
   AxisRun.Axis[11].Pos6.Position := 0.0;
   AxisRun.Axis[11].Pos6.Speed := 0;
   AxisRun.Axis[11].Pos6.Reached := FALSE;
   AxisRun.Axis[11].Pos7.Position := 0.0;
   AxisRun.Axis[11].Pos7.Speed := 0;
   AxisRun.Axis[11].Pos7.Reached := FALSE;
   AxisRun.Axis[11].Pos8.Position := 0.0;
   AxisRun.Axis[11].Pos8.Speed := 0;
   AxisRun.Axis[11].Pos8.Reached := FALSE;
   AxisRun.Axis[11].Pos9.Position := 0.0;
   AxisRun.Axis[11].Pos9.Speed := 0;
   AxisRun.Axis[11].Pos9.Reached := FALSE;
   AxisRun.Axis[11].Pos10.Position := 0.0;
   AxisRun.Axis[11].Pos10.Speed := 0;
   AxisRun.Axis[11].Pos10.Reached := FALSE;
   AxisRun.Axis[11].Pos11.Position := 0.0;
   AxisRun.Axis[11].Pos11.Speed := 0;
   AxisRun.Axis[11].Pos11.Reached := FALSE;
   AxisRun.Axis[11].Pos12.Position := 0.0;
   AxisRun.Axis[11].Pos12.Speed := 0;
   AxisRun.Axis[11].Pos12.Reached := FALSE;
   AxisRun.Axis[11].Pos13.Position := 0.0;
   AxisRun.Axis[11].Pos13.Speed := 0;
   AxisRun.Axis[11].Pos13.Reached := FALSE;
   AxisRun.Axis[11].Pos14.Position := 0.0;
   AxisRun.Axis[11].Pos14.Speed := 0;
   AxisRun.Axis[11].Pos14.Reached := FALSE;
   AxisRun.Axis[11].Pos15.Position := 0.0;
   AxisRun.Axis[11].Pos15.Speed := 0;
   AxisRun.Axis[11].Pos15.Reached := FALSE;
   AxisRun.Axis[11].Pos16.Position := 0.0;
   AxisRun.Axis[11].Pos16.Speed := 0;
   AxisRun.Axis[11].Pos16.Reached := FALSE;
   AxisRun.Axis[11].Pos17.Position := 0.0;
   AxisRun.Axis[11].Pos17.Speed := 0;
   AxisRun.Axis[11].Pos17.Reached := FALSE;
   AxisRun.Axis[11].Pos18.Position := 0.0;
   AxisRun.Axis[11].Pos18.Speed := 0;
   AxisRun.Axis[11].Pos18.Reached := FALSE;
   AxisRun.Axis[11].Pos19.Position := 0.0;
   AxisRun.Axis[11].Pos19.Speed := 0;
   AxisRun.Axis[11].Pos19.Reached := FALSE;
   AxisRun.Axis[11].Pos20.Position := 0.0;
   AxisRun.Axis[11].Pos20.Speed := 0;
   AxisRun.Axis[11].Pos20.Reached := FALSE;
   AxisRun.Axis[11].Pos21.Position := 0.0;
   AxisRun.Axis[11].Pos21.Speed := 0;
   AxisRun.Axis[11].Pos21.Reached := FALSE;
   AxisRun.Axis[11].Pos22.Position := 0.0;
   AxisRun.Axis[11].Pos22.Speed := 0;
   AxisRun.Axis[11].Pos22.Reached := FALSE;
   AxisRun.Axis[11].Pos23.Position := 0.0;
   AxisRun.Axis[11].Pos23.Speed := 0;
   AxisRun.Axis[11].Pos23.Reached := FALSE;
   AxisRun.Axis[11].Pos24.Position := 0.0;
   AxisRun.Axis[11].Pos24.Speed := 0;
   AxisRun.Axis[11].Pos24.Reached := FALSE;
   AxisRun.Axis[11].Pos25.Position := 0.0;
   AxisRun.Axis[11].Pos25.Speed := 0;
   AxisRun.Axis[11].Pos25.Reached := FALSE;
   AxisRun.Axis[11].Pos26.Position := 0.0;
   AxisRun.Axis[11].Pos26.Speed := 0;
   AxisRun.Axis[11].Pos26.Reached := FALSE;
   AxisRun.Axis[11].Pos27.Position := 0.0;
   AxisRun.Axis[11].Pos27.Speed := 0;
   AxisRun.Axis[11].Pos27.Reached := FALSE;
   AxisRun.Axis[11].Pos28.Position := 0.0;
   AxisRun.Axis[11].Pos28.Speed := 0;
   AxisRun.Axis[11].Pos28.Reached := FALSE;
   AxisRun.Axis[11].Pos29.Position := 0.0;
   AxisRun.Axis[11].Pos29.Speed := 0;
   AxisRun.Axis[11].Pos29.Reached := FALSE;
   AxisRun.Axis[11].Pos30.Position := 0.0;
   AxisRun.Axis[11].Pos30.Speed := 0;
   AxisRun.Axis[11].Pos30.Reached := FALSE;
   AxisRun.Axis[12].Pos1.Position := 0.0;
   AxisRun.Axis[12].Pos1.Speed := 0;
   AxisRun.Axis[12].Pos1.Reached := FALSE;
   AxisRun.Axis[12].Pos2.Position := 0.0;
   AxisRun.Axis[12].Pos2.Speed := 0;
   AxisRun.Axis[12].Pos2.Reached := FALSE;
   AxisRun.Axis[12].Pos3.Position := 0.0;
   AxisRun.Axis[12].Pos3.Speed := 0;
   AxisRun.Axis[12].Pos3.Reached := FALSE;
   AxisRun.Axis[12].Pos4.Position := 0.0;
   AxisRun.Axis[12].Pos4.Speed := 0;
   AxisRun.Axis[12].Pos4.Reached := FALSE;
   AxisRun.Axis[12].Pos5.Position := 0.0;
   AxisRun.Axis[12].Pos5.Speed := 0;
   AxisRun.Axis[12].Pos5.Reached := FALSE;
   AxisRun.Axis[12].Pos6.Position := 0.0;
   AxisRun.Axis[12].Pos6.Speed := 0;
   AxisRun.Axis[12].Pos6.Reached := FALSE;
   AxisRun.Axis[12].Pos7.Position := 0.0;
   AxisRun.Axis[12].Pos7.Speed := 0;
   AxisRun.Axis[12].Pos7.Reached := FALSE;
   AxisRun.Axis[12].Pos8.Position := 0.0;
   AxisRun.Axis[12].Pos8.Speed := 0;
   AxisRun.Axis[12].Pos8.Reached := FALSE;
   AxisRun.Axis[12].Pos9.Position := 0.0;
   AxisRun.Axis[12].Pos9.Speed := 0;
   AxisRun.Axis[12].Pos9.Reached := FALSE;
   AxisRun.Axis[12].Pos10.Position := 0.0;
   AxisRun.Axis[12].Pos10.Speed := 0;
   AxisRun.Axis[12].Pos10.Reached := FALSE;
   AxisRun.Axis[12].Pos11.Position := 0.0;
   AxisRun.Axis[12].Pos11.Speed := 0;
   AxisRun.Axis[12].Pos11.Reached := FALSE;
   AxisRun.Axis[12].Pos12.Position := 0.0;
   AxisRun.Axis[12].Pos12.Speed := 0;
   AxisRun.Axis[12].Pos12.Reached := FALSE;
   AxisRun.Axis[12].Pos13.Position := 0.0;
   AxisRun.Axis[12].Pos13.Speed := 0;
   AxisRun.Axis[12].Pos13.Reached := FALSE;
   AxisRun.Axis[12].Pos14.Position := 0.0;
   AxisRun.Axis[12].Pos14.Speed := 0;
   AxisRun.Axis[12].Pos14.Reached := FALSE;
   AxisRun.Axis[12].Pos15.Position := 0.0;
   AxisRun.Axis[12].Pos15.Speed := 0;
   AxisRun.Axis[12].Pos15.Reached := FALSE;
   AxisRun.Axis[12].Pos16.Position := 0.0;
   AxisRun.Axis[12].Pos16.Speed := 0;
   AxisRun.Axis[12].Pos16.Reached := FALSE;
   AxisRun.Axis[12].Pos17.Position := 0.0;
   AxisRun.Axis[12].Pos17.Speed := 0;
   AxisRun.Axis[12].Pos17.Reached := FALSE;
   AxisRun.Axis[12].Pos18.Position := 0.0;
   AxisRun.Axis[12].Pos18.Speed := 0;
   AxisRun.Axis[12].Pos18.Reached := FALSE;
   AxisRun.Axis[12].Pos19.Position := 0.0;
   AxisRun.Axis[12].Pos19.Speed := 0;
   AxisRun.Axis[12].Pos19.Reached := FALSE;
   AxisRun.Axis[12].Pos20.Position := 0.0;
   AxisRun.Axis[12].Pos20.Speed := 0;
   AxisRun.Axis[12].Pos20.Reached := FALSE;
   AxisRun.Axis[12].Pos21.Position := 0.0;
   AxisRun.Axis[12].Pos21.Speed := 0;
   AxisRun.Axis[12].Pos21.Reached := FALSE;
   AxisRun.Axis[12].Pos22.Position := 0.0;
   AxisRun.Axis[12].Pos22.Speed := 0;
   AxisRun.Axis[12].Pos22.Reached := FALSE;
   AxisRun.Axis[12].Pos23.Position := 0.0;
   AxisRun.Axis[12].Pos23.Speed := 0;
   AxisRun.Axis[12].Pos23.Reached := FALSE;
   AxisRun.Axis[12].Pos24.Position := 0.0;
   AxisRun.Axis[12].Pos24.Speed := 0;
   AxisRun.Axis[12].Pos24.Reached := FALSE;
   AxisRun.Axis[12].Pos25.Position := 0.0;
   AxisRun.Axis[12].Pos25.Speed := 0;
   AxisRun.Axis[12].Pos25.Reached := FALSE;
   AxisRun.Axis[12].Pos26.Position := 0.0;
   AxisRun.Axis[12].Pos26.Speed := 0;
   AxisRun.Axis[12].Pos26.Reached := FALSE;
   AxisRun.Axis[12].Pos27.Position := 0.0;
   AxisRun.Axis[12].Pos27.Speed := 0;
   AxisRun.Axis[12].Pos27.Reached := FALSE;
   AxisRun.Axis[12].Pos28.Position := 0.0;
   AxisRun.Axis[12].Pos28.Speed := 0;
   AxisRun.Axis[12].Pos28.Reached := FALSE;
   AxisRun.Axis[12].Pos29.Position := 0.0;
   AxisRun.Axis[12].Pos29.Speed := 0;
   AxisRun.Axis[12].Pos29.Reached := FALSE;
   AxisRun.Axis[12].Pos30.Position := 0.0;
   AxisRun.Axis[12].Pos30.Speed := 0;
   AxisRun.Axis[12].Pos30.Reached := FALSE;
   AxisRun.Axis[13].Pos1.Position := 0.0;
   AxisRun.Axis[13].Pos1.Speed := 0;
   AxisRun.Axis[13].Pos1.Reached := FALSE;
   AxisRun.Axis[13].Pos2.Position := 0.0;
   AxisRun.Axis[13].Pos2.Speed := 0;
   AxisRun.Axis[13].Pos2.Reached := FALSE;
   AxisRun.Axis[13].Pos3.Position := 0.0;
   AxisRun.Axis[13].Pos3.Speed := 0;
   AxisRun.Axis[13].Pos3.Reached := FALSE;
   AxisRun.Axis[13].Pos4.Position := 0.0;
   AxisRun.Axis[13].Pos4.Speed := 0;
   AxisRun.Axis[13].Pos4.Reached := FALSE;
   AxisRun.Axis[13].Pos5.Position := 0.0;
   AxisRun.Axis[13].Pos5.Speed := 0;
   AxisRun.Axis[13].Pos5.Reached := FALSE;
   AxisRun.Axis[13].Pos6.Position := 0.0;
   AxisRun.Axis[13].Pos6.Speed := 0;
   AxisRun.Axis[13].Pos6.Reached := FALSE;
   AxisRun.Axis[13].Pos7.Position := 0.0;
   AxisRun.Axis[13].Pos7.Speed := 0;
   AxisRun.Axis[13].Pos7.Reached := FALSE;
   AxisRun.Axis[13].Pos8.Position := 0.0;
   AxisRun.Axis[13].Pos8.Speed := 0;
   AxisRun.Axis[13].Pos8.Reached := FALSE;
   AxisRun.Axis[13].Pos9.Position := 0.0;
   AxisRun.Axis[13].Pos9.Speed := 0;
   AxisRun.Axis[13].Pos9.Reached := FALSE;
   AxisRun.Axis[13].Pos10.Position := 0.0;
   AxisRun.Axis[13].Pos10.Speed := 0;
   AxisRun.Axis[13].Pos10.Reached := FALSE;
   AxisRun.Axis[13].Pos11.Position := 0.0;
   AxisRun.Axis[13].Pos11.Speed := 0;
   AxisRun.Axis[13].Pos11.Reached := FALSE;
   AxisRun.Axis[13].Pos12.Position := 0.0;
   AxisRun.Axis[13].Pos12.Speed := 0;
   AxisRun.Axis[13].Pos12.Reached := FALSE;
   AxisRun.Axis[13].Pos13.Position := 0.0;
   AxisRun.Axis[13].Pos13.Speed := 0;
   AxisRun.Axis[13].Pos13.Reached := FALSE;
   AxisRun.Axis[13].Pos14.Position := 0.0;
   AxisRun.Axis[13].Pos14.Speed := 0;
   AxisRun.Axis[13].Pos14.Reached := FALSE;
   AxisRun.Axis[13].Pos15.Position := 0.0;
   AxisRun.Axis[13].Pos15.Speed := 0;
   AxisRun.Axis[13].Pos15.Reached := FALSE;
   AxisRun.Axis[13].Pos16.Position := 0.0;
   AxisRun.Axis[13].Pos16.Speed := 0;
   AxisRun.Axis[13].Pos16.Reached := FALSE;
   AxisRun.Axis[13].Pos17.Position := 0.0;
   AxisRun.Axis[13].Pos17.Speed := 0;
   AxisRun.Axis[13].Pos17.Reached := FALSE;
   AxisRun.Axis[13].Pos18.Position := 0.0;
   AxisRun.Axis[13].Pos18.Speed := 0;
   AxisRun.Axis[13].Pos18.Reached := FALSE;
   AxisRun.Axis[13].Pos19.Position := 0.0;
   AxisRun.Axis[13].Pos19.Speed := 0;
   AxisRun.Axis[13].Pos19.Reached := FALSE;
   AxisRun.Axis[13].Pos20.Position := 0.0;
   AxisRun.Axis[13].Pos20.Speed := 0;
   AxisRun.Axis[13].Pos20.Reached := FALSE;
   AxisRun.Axis[13].Pos21.Position := 0.0;
   AxisRun.Axis[13].Pos21.Speed := 0;
   AxisRun.Axis[13].Pos21.Reached := FALSE;
   AxisRun.Axis[13].Pos22.Position := 0.0;
   AxisRun.Axis[13].Pos22.Speed := 0;
   AxisRun.Axis[13].Pos22.Reached := FALSE;
   AxisRun.Axis[13].Pos23.Position := 0.0;
   AxisRun.Axis[13].Pos23.Speed := 0;
   AxisRun.Axis[13].Pos23.Reached := FALSE;
   AxisRun.Axis[13].Pos24.Position := 0.0;
   AxisRun.Axis[13].Pos24.Speed := 0;
   AxisRun.Axis[13].Pos24.Reached := FALSE;
   AxisRun.Axis[13].Pos25.Position := 0.0;
   AxisRun.Axis[13].Pos25.Speed := 0;
   AxisRun.Axis[13].Pos25.Reached := FALSE;
   AxisRun.Axis[13].Pos26.Position := 0.0;
   AxisRun.Axis[13].Pos26.Speed := 0;
   AxisRun.Axis[13].Pos26.Reached := FALSE;
   AxisRun.Axis[13].Pos27.Position := 0.0;
   AxisRun.Axis[13].Pos27.Speed := 0;
   AxisRun.Axis[13].Pos27.Reached := FALSE;
   AxisRun.Axis[13].Pos28.Position := 0.0;
   AxisRun.Axis[13].Pos28.Speed := 0;
   AxisRun.Axis[13].Pos28.Reached := FALSE;
   AxisRun.Axis[13].Pos29.Position := 0.0;
   AxisRun.Axis[13].Pos29.Speed := 0;
   AxisRun.Axis[13].Pos29.Reached := FALSE;
   AxisRun.Axis[13].Pos30.Position := 0.0;
   AxisRun.Axis[13].Pos30.Speed := 0;
   AxisRun.Axis[13].Pos30.Reached := FALSE;
   AxisRun.Axis[14].Pos1.Position := 0.0;
   AxisRun.Axis[14].Pos1.Speed := 0;
   AxisRun.Axis[14].Pos1.Reached := FALSE;
   AxisRun.Axis[14].Pos2.Position := 0.0;
   AxisRun.Axis[14].Pos2.Speed := 0;
   AxisRun.Axis[14].Pos2.Reached := FALSE;
   AxisRun.Axis[14].Pos3.Position := 0.0;
   AxisRun.Axis[14].Pos3.Speed := 0;
   AxisRun.Axis[14].Pos3.Reached := FALSE;
   AxisRun.Axis[14].Pos4.Position := 0.0;
   AxisRun.Axis[14].Pos4.Speed := 0;
   AxisRun.Axis[14].Pos4.Reached := FALSE;
   AxisRun.Axis[14].Pos5.Position := 0.0;
   AxisRun.Axis[14].Pos5.Speed := 0;
   AxisRun.Axis[14].Pos5.Reached := FALSE;
   AxisRun.Axis[14].Pos6.Position := 0.0;
   AxisRun.Axis[14].Pos6.Speed := 0;
   AxisRun.Axis[14].Pos6.Reached := FALSE;
   AxisRun.Axis[14].Pos7.Position := 0.0;
   AxisRun.Axis[14].Pos7.Speed := 0;
   AxisRun.Axis[14].Pos7.Reached := FALSE;
   AxisRun.Axis[14].Pos8.Position := 0.0;
   AxisRun.Axis[14].Pos8.Speed := 0;
   AxisRun.Axis[14].Pos8.Reached := FALSE;
   AxisRun.Axis[14].Pos9.Position := 0.0;
   AxisRun.Axis[14].Pos9.Speed := 0;
   AxisRun.Axis[14].Pos9.Reached := FALSE;
   AxisRun.Axis[14].Pos10.Position := 0.0;
   AxisRun.Axis[14].Pos10.Speed := 0;
   AxisRun.Axis[14].Pos10.Reached := FALSE;
   AxisRun.Axis[14].Pos11.Position := 0.0;
   AxisRun.Axis[14].Pos11.Speed := 0;
   AxisRun.Axis[14].Pos11.Reached := FALSE;
   AxisRun.Axis[14].Pos12.Position := 0.0;
   AxisRun.Axis[14].Pos12.Speed := 0;
   AxisRun.Axis[14].Pos12.Reached := FALSE;
   AxisRun.Axis[14].Pos13.Position := 0.0;
   AxisRun.Axis[14].Pos13.Speed := 0;
   AxisRun.Axis[14].Pos13.Reached := FALSE;
   AxisRun.Axis[14].Pos14.Position := 0.0;
   AxisRun.Axis[14].Pos14.Speed := 0;
   AxisRun.Axis[14].Pos14.Reached := FALSE;
   AxisRun.Axis[14].Pos15.Position := 0.0;
   AxisRun.Axis[14].Pos15.Speed := 0;
   AxisRun.Axis[14].Pos15.Reached := FALSE;
   AxisRun.Axis[14].Pos16.Position := 0.0;
   AxisRun.Axis[14].Pos16.Speed := 0;
   AxisRun.Axis[14].Pos16.Reached := FALSE;
   AxisRun.Axis[14].Pos17.Position := 0.0;
   AxisRun.Axis[14].Pos17.Speed := 0;
   AxisRun.Axis[14].Pos17.Reached := FALSE;
   AxisRun.Axis[14].Pos18.Position := 0.0;
   AxisRun.Axis[14].Pos18.Speed := 0;
   AxisRun.Axis[14].Pos18.Reached := FALSE;
   AxisRun.Axis[14].Pos19.Position := 0.0;
   AxisRun.Axis[14].Pos19.Speed := 0;
   AxisRun.Axis[14].Pos19.Reached := FALSE;
   AxisRun.Axis[14].Pos20.Position := 0.0;
   AxisRun.Axis[14].Pos20.Speed := 0;
   AxisRun.Axis[14].Pos20.Reached := FALSE;
   AxisRun.Axis[14].Pos21.Position := 0.0;
   AxisRun.Axis[14].Pos21.Speed := 0;
   AxisRun.Axis[14].Pos21.Reached := FALSE;
   AxisRun.Axis[14].Pos22.Position := 0.0;
   AxisRun.Axis[14].Pos22.Speed := 0;
   AxisRun.Axis[14].Pos22.Reached := FALSE;
   AxisRun.Axis[14].Pos23.Position := 0.0;
   AxisRun.Axis[14].Pos23.Speed := 0;
   AxisRun.Axis[14].Pos23.Reached := FALSE;
   AxisRun.Axis[14].Pos24.Position := 0.0;
   AxisRun.Axis[14].Pos24.Speed := 0;
   AxisRun.Axis[14].Pos24.Reached := FALSE;
   AxisRun.Axis[14].Pos25.Position := 0.0;
   AxisRun.Axis[14].Pos25.Speed := 0;
   AxisRun.Axis[14].Pos25.Reached := FALSE;
   AxisRun.Axis[14].Pos26.Position := 0.0;
   AxisRun.Axis[14].Pos26.Speed := 0;
   AxisRun.Axis[14].Pos26.Reached := FALSE;
   AxisRun.Axis[14].Pos27.Position := 0.0;
   AxisRun.Axis[14].Pos27.Speed := 0;
   AxisRun.Axis[14].Pos27.Reached := FALSE;
   AxisRun.Axis[14].Pos28.Position := 0.0;
   AxisRun.Axis[14].Pos28.Speed := 0;
   AxisRun.Axis[14].Pos28.Reached := FALSE;
   AxisRun.Axis[14].Pos29.Position := 0.0;
   AxisRun.Axis[14].Pos29.Speed := 0;
   AxisRun.Axis[14].Pos29.Reached := FALSE;
   AxisRun.Axis[14].Pos30.Position := 0.0;
   AxisRun.Axis[14].Pos30.Speed := 0;
   AxisRun.Axis[14].Pos30.Reached := FALSE;
   AxisRun.Axis[15].Pos1.Position := 0.0;
   AxisRun.Axis[15].Pos1.Speed := 0;
   AxisRun.Axis[15].Pos1.Reached := FALSE;
   AxisRun.Axis[15].Pos2.Position := 0.0;
   AxisRun.Axis[15].Pos2.Speed := 0;
   AxisRun.Axis[15].Pos2.Reached := FALSE;
   AxisRun.Axis[15].Pos3.Position := 0.0;
   AxisRun.Axis[15].Pos3.Speed := 0;
   AxisRun.Axis[15].Pos3.Reached := FALSE;
   AxisRun.Axis[15].Pos4.Position := 0.0;
   AxisRun.Axis[15].Pos4.Speed := 0;
   AxisRun.Axis[15].Pos4.Reached := FALSE;
   AxisRun.Axis[15].Pos5.Position := 0.0;
   AxisRun.Axis[15].Pos5.Speed := 0;
   AxisRun.Axis[15].Pos5.Reached := FALSE;
   AxisRun.Axis[15].Pos6.Position := 0.0;
   AxisRun.Axis[15].Pos6.Speed := 0;
   AxisRun.Axis[15].Pos6.Reached := FALSE;
   AxisRun.Axis[15].Pos7.Position := 0.0;
   AxisRun.Axis[15].Pos7.Speed := 0;
   AxisRun.Axis[15].Pos7.Reached := FALSE;
   AxisRun.Axis[15].Pos8.Position := 0.0;
   AxisRun.Axis[15].Pos8.Speed := 0;
   AxisRun.Axis[15].Pos8.Reached := FALSE;
   AxisRun.Axis[15].Pos9.Position := 0.0;
   AxisRun.Axis[15].Pos9.Speed := 0;
   AxisRun.Axis[15].Pos9.Reached := FALSE;
   AxisRun.Axis[15].Pos10.Position := 0.0;
   AxisRun.Axis[15].Pos10.Speed := 0;
   AxisRun.Axis[15].Pos10.Reached := FALSE;
   AxisRun.Axis[15].Pos11.Position := 0.0;
   AxisRun.Axis[15].Pos11.Speed := 0;
   AxisRun.Axis[15].Pos11.Reached := FALSE;
   AxisRun.Axis[15].Pos12.Position := 0.0;
   AxisRun.Axis[15].Pos12.Speed := 0;
   AxisRun.Axis[15].Pos12.Reached := FALSE;
   AxisRun.Axis[15].Pos13.Position := 0.0;
   AxisRun.Axis[15].Pos13.Speed := 0;
   AxisRun.Axis[15].Pos13.Reached := FALSE;
   AxisRun.Axis[15].Pos14.Position := 0.0;
   AxisRun.Axis[15].Pos14.Speed := 0;
   AxisRun.Axis[15].Pos14.Reached := FALSE;
   AxisRun.Axis[15].Pos15.Position := 0.0;
   AxisRun.Axis[15].Pos15.Speed := 0;
   AxisRun.Axis[15].Pos15.Reached := FALSE;
   AxisRun.Axis[15].Pos16.Position := 0.0;
   AxisRun.Axis[15].Pos16.Speed := 0;
   AxisRun.Axis[15].Pos16.Reached := FALSE;
   AxisRun.Axis[15].Pos17.Position := 0.0;
   AxisRun.Axis[15].Pos17.Speed := 0;
   AxisRun.Axis[15].Pos17.Reached := FALSE;
   AxisRun.Axis[15].Pos18.Position := 0.0;
   AxisRun.Axis[15].Pos18.Speed := 0;
   AxisRun.Axis[15].Pos18.Reached := FALSE;
   AxisRun.Axis[15].Pos19.Position := 0.0;
   AxisRun.Axis[15].Pos19.Speed := 0;
   AxisRun.Axis[15].Pos19.Reached := FALSE;
   AxisRun.Axis[15].Pos20.Position := 0.0;
   AxisRun.Axis[15].Pos20.Speed := 0;
   AxisRun.Axis[15].Pos20.Reached := FALSE;
   AxisRun.Axis[15].Pos21.Position := 0.0;
   AxisRun.Axis[15].Pos21.Speed := 0;
   AxisRun.Axis[15].Pos21.Reached := FALSE;
   AxisRun.Axis[15].Pos22.Position := 0.0;
   AxisRun.Axis[15].Pos22.Speed := 0;
   AxisRun.Axis[15].Pos22.Reached := FALSE;
   AxisRun.Axis[15].Pos23.Position := 0.0;
   AxisRun.Axis[15].Pos23.Speed := 0;
   AxisRun.Axis[15].Pos23.Reached := FALSE;
   AxisRun.Axis[15].Pos24.Position := 0.0;
   AxisRun.Axis[15].Pos24.Speed := 0;
   AxisRun.Axis[15].Pos24.Reached := FALSE;
   AxisRun.Axis[15].Pos25.Position := 0.0;
   AxisRun.Axis[15].Pos25.Speed := 0;
   AxisRun.Axis[15].Pos25.Reached := FALSE;
   AxisRun.Axis[15].Pos26.Position := 0.0;
   AxisRun.Axis[15].Pos26.Speed := 0;
   AxisRun.Axis[15].Pos26.Reached := FALSE;
   AxisRun.Axis[15].Pos27.Position := 0.0;
   AxisRun.Axis[15].Pos27.Speed := 0;
   AxisRun.Axis[15].Pos27.Reached := FALSE;
   AxisRun.Axis[15].Pos28.Position := 0.0;
   AxisRun.Axis[15].Pos28.Speed := 0;
   AxisRun.Axis[15].Pos28.Reached := FALSE;
   AxisRun.Axis[15].Pos29.Position := 0.0;
   AxisRun.Axis[15].Pos29.Speed := 0;
   AxisRun.Axis[15].Pos29.Reached := FALSE;
   AxisRun.Axis[15].Pos30.Position := 0.0;
   AxisRun.Axis[15].Pos30.Speed := 0;
   AxisRun.Axis[15].Pos30.Reached := FALSE;
   AxisNuw.Axis[1].Pos1.Position := 0.0;
   AxisNuw.Axis[1].Pos1.Speed := 0;
   AxisNuw.Axis[1].Pos1.Reached := FALSE;
   AxisNuw.Axis[1].Pos2.Position := 0.0;
   AxisNuw.Axis[1].Pos2.Speed := 0;
   AxisNuw.Axis[1].Pos2.Reached := FALSE;
   AxisNuw.Axis[1].Pos3.Position := 0.0;
   AxisNuw.Axis[1].Pos3.Speed := 0;
   AxisNuw.Axis[1].Pos3.Reached := FALSE;
   AxisNuw.Axis[1].Pos4.Position := 0.0;
   AxisNuw.Axis[1].Pos4.Speed := 0;
   AxisNuw.Axis[1].Pos4.Reached := FALSE;
   AxisNuw.Axis[1].Pos5.Position := 0.0;
   AxisNuw.Axis[1].Pos5.Speed := 0;
   AxisNuw.Axis[1].Pos5.Reached := FALSE;
   AxisNuw.Axis[1].Pos6.Position := 0.0;
   AxisNuw.Axis[1].Pos6.Speed := 0;
   AxisNuw.Axis[1].Pos6.Reached := FALSE;
   AxisNuw.Axis[1].Pos7.Position := 0.0;
   AxisNuw.Axis[1].Pos7.Speed := 0;
   AxisNuw.Axis[1].Pos7.Reached := FALSE;
   AxisNuw.Axis[1].Pos8.Position := 0.0;
   AxisNuw.Axis[1].Pos8.Speed := 0;
   AxisNuw.Axis[1].Pos8.Reached := FALSE;
   AxisNuw.Axis[1].Pos9.Position := 0.0;
   AxisNuw.Axis[1].Pos9.Speed := 0;
   AxisNuw.Axis[1].Pos9.Reached := FALSE;
   AxisNuw.Axis[1].Pos10.Position := 0.0;
   AxisNuw.Axis[1].Pos10.Speed := 0;
   AxisNuw.Axis[1].Pos10.Reached := FALSE;
   AxisNuw.Axis[1].Pos11.Position := 0.0;
   AxisNuw.Axis[1].Pos11.Speed := 0;
   AxisNuw.Axis[1].Pos11.Reached := FALSE;
   AxisNuw.Axis[1].Pos12.Position := 0.0;
   AxisNuw.Axis[1].Pos12.Speed := 0;
   AxisNuw.Axis[1].Pos12.Reached := FALSE;
   AxisNuw.Axis[1].Pos13.Position := 0.0;
   AxisNuw.Axis[1].Pos13.Speed := 0;
   AxisNuw.Axis[1].Pos13.Reached := FALSE;
   AxisNuw.Axis[1].Pos14.Position := 0.0;
   AxisNuw.Axis[1].Pos14.Speed := 0;
   AxisNuw.Axis[1].Pos14.Reached := FALSE;
   AxisNuw.Axis[1].Pos15.Position := 0.0;
   AxisNuw.Axis[1].Pos15.Speed := 0;
   AxisNuw.Axis[1].Pos15.Reached := FALSE;
   AxisNuw.Axis[1].Pos16.Position := 0.0;
   AxisNuw.Axis[1].Pos16.Speed := 0;
   AxisNuw.Axis[1].Pos16.Reached := FALSE;
   AxisNuw.Axis[1].Pos17.Position := 0.0;
   AxisNuw.Axis[1].Pos17.Speed := 0;
   AxisNuw.Axis[1].Pos17.Reached := FALSE;
   AxisNuw.Axis[1].Pos18.Position := 0.0;
   AxisNuw.Axis[1].Pos18.Speed := 0;
   AxisNuw.Axis[1].Pos18.Reached := FALSE;
   AxisNuw.Axis[1].Pos19.Position := 0.0;
   AxisNuw.Axis[1].Pos19.Speed := 0;
   AxisNuw.Axis[1].Pos19.Reached := FALSE;
   AxisNuw.Axis[1].Pos20.Position := 0.0;
   AxisNuw.Axis[1].Pos20.Speed := 0;
   AxisNuw.Axis[1].Pos20.Reached := FALSE;
   AxisNuw.Axis[1].Pos21.Position := 0.0;
   AxisNuw.Axis[1].Pos21.Speed := 0;
   AxisNuw.Axis[1].Pos21.Reached := FALSE;
   AxisNuw.Axis[1].Pos22.Position := 0.0;
   AxisNuw.Axis[1].Pos22.Speed := 0;
   AxisNuw.Axis[1].Pos22.Reached := FALSE;
   AxisNuw.Axis[1].Pos23.Position := 0.0;
   AxisNuw.Axis[1].Pos23.Speed := 0;
   AxisNuw.Axis[1].Pos23.Reached := FALSE;
   AxisNuw.Axis[1].Pos24.Position := 0.0;
   AxisNuw.Axis[1].Pos24.Speed := 0;
   AxisNuw.Axis[1].Pos24.Reached := FALSE;
   AxisNuw.Axis[1].Pos25.Position := 0.0;
   AxisNuw.Axis[1].Pos25.Speed := 0;
   AxisNuw.Axis[1].Pos25.Reached := FALSE;
   AxisNuw.Axis[1].Pos26.Position := 0.0;
   AxisNuw.Axis[1].Pos26.Speed := 0;
   AxisNuw.Axis[1].Pos26.Reached := FALSE;
   AxisNuw.Axis[1].Pos27.Position := 0.0;
   AxisNuw.Axis[1].Pos27.Speed := 0;
   AxisNuw.Axis[1].Pos27.Reached := FALSE;
   AxisNuw.Axis[1].Pos28.Position := 0.0;
   AxisNuw.Axis[1].Pos28.Speed := 0;
   AxisNuw.Axis[1].Pos28.Reached := FALSE;
   AxisNuw.Axis[1].Pos29.Position := 0.0;
   AxisNuw.Axis[1].Pos29.Speed := 0;
   AxisNuw.Axis[1].Pos29.Reached := FALSE;
   AxisNuw.Axis[1].Pos30.Position := 0.0;
   AxisNuw.Axis[1].Pos30.Speed := 0;
   AxisNuw.Axis[1].Pos30.Reached := FALSE;
   AxisNuw.Axis[2].Pos1.Position := 0.0;
   AxisNuw.Axis[2].Pos1.Speed := 0;
   AxisNuw.Axis[2].Pos1.Reached := FALSE;
   AxisNuw.Axis[2].Pos2.Position := 0.0;
   AxisNuw.Axis[2].Pos2.Speed := 0;
   AxisNuw.Axis[2].Pos2.Reached := FALSE;
   AxisNuw.Axis[2].Pos3.Position := 0.0;
   AxisNuw.Axis[2].Pos3.Speed := 0;
   AxisNuw.Axis[2].Pos3.Reached := FALSE;
   AxisNuw.Axis[2].Pos4.Position := 0.0;
   AxisNuw.Axis[2].Pos4.Speed := 0;
   AxisNuw.Axis[2].Pos4.Reached := FALSE;
   AxisNuw.Axis[2].Pos5.Position := 0.0;
   AxisNuw.Axis[2].Pos5.Speed := 0;
   AxisNuw.Axis[2].Pos5.Reached := FALSE;
   AxisNuw.Axis[2].Pos6.Position := 0.0;
   AxisNuw.Axis[2].Pos6.Speed := 0;
   AxisNuw.Axis[2].Pos6.Reached := FALSE;
   AxisNuw.Axis[2].Pos7.Position := 0.0;
   AxisNuw.Axis[2].Pos7.Speed := 0;
   AxisNuw.Axis[2].Pos7.Reached := FALSE;
   AxisNuw.Axis[2].Pos8.Position := 0.0;
   AxisNuw.Axis[2].Pos8.Speed := 0;
   AxisNuw.Axis[2].Pos8.Reached := FALSE;
   AxisNuw.Axis[2].Pos9.Position := 0.0;
   AxisNuw.Axis[2].Pos9.Speed := 0;
   AxisNuw.Axis[2].Pos9.Reached := FALSE;
   AxisNuw.Axis[2].Pos10.Position := 0.0;
   AxisNuw.Axis[2].Pos10.Speed := 0;
   AxisNuw.Axis[2].Pos10.Reached := FALSE;
   AxisNuw.Axis[2].Pos11.Position := 0.0;
   AxisNuw.Axis[2].Pos11.Speed := 0;
   AxisNuw.Axis[2].Pos11.Reached := FALSE;
   AxisNuw.Axis[2].Pos12.Position := 0.0;
   AxisNuw.Axis[2].Pos12.Speed := 0;
   AxisNuw.Axis[2].Pos12.Reached := FALSE;
   AxisNuw.Axis[2].Pos13.Position := 0.0;
   AxisNuw.Axis[2].Pos13.Speed := 0;
   AxisNuw.Axis[2].Pos13.Reached := FALSE;
   AxisNuw.Axis[2].Pos14.Position := 0.0;
   AxisNuw.Axis[2].Pos14.Speed := 0;
   AxisNuw.Axis[2].Pos14.Reached := FALSE;
   AxisNuw.Axis[2].Pos15.Position := 0.0;
   AxisNuw.Axis[2].Pos15.Speed := 0;
   AxisNuw.Axis[2].Pos15.Reached := FALSE;
   AxisNuw.Axis[2].Pos16.Position := 0.0;
   AxisNuw.Axis[2].Pos16.Speed := 0;
   AxisNuw.Axis[2].Pos16.Reached := FALSE;
   AxisNuw.Axis[2].Pos17.Position := 0.0;
   AxisNuw.Axis[2].Pos17.Speed := 0;
   AxisNuw.Axis[2].Pos17.Reached := FALSE;
   AxisNuw.Axis[2].Pos18.Position := 0.0;
   AxisNuw.Axis[2].Pos18.Speed := 0;
   AxisNuw.Axis[2].Pos18.Reached := FALSE;
   AxisNuw.Axis[2].Pos19.Position := 0.0;
   AxisNuw.Axis[2].Pos19.Speed := 0;
   AxisNuw.Axis[2].Pos19.Reached := FALSE;
   AxisNuw.Axis[2].Pos20.Position := 0.0;
   AxisNuw.Axis[2].Pos20.Speed := 0;
   AxisNuw.Axis[2].Pos20.Reached := FALSE;
   AxisNuw.Axis[2].Pos21.Position := 0.0;
   AxisNuw.Axis[2].Pos21.Speed := 0;
   AxisNuw.Axis[2].Pos21.Reached := FALSE;
   AxisNuw.Axis[2].Pos22.Position := 0.0;
   AxisNuw.Axis[2].Pos22.Speed := 0;
   AxisNuw.Axis[2].Pos22.Reached := FALSE;
   AxisNuw.Axis[2].Pos23.Position := 0.0;
   AxisNuw.Axis[2].Pos23.Speed := 0;
   AxisNuw.Axis[2].Pos23.Reached := FALSE;
   AxisNuw.Axis[2].Pos24.Position := 0.0;
   AxisNuw.Axis[2].Pos24.Speed := 0;
   AxisNuw.Axis[2].Pos24.Reached := FALSE;
   AxisNuw.Axis[2].Pos25.Position := 0.0;
   AxisNuw.Axis[2].Pos25.Speed := 0;
   AxisNuw.Axis[2].Pos25.Reached := FALSE;
   AxisNuw.Axis[2].Pos26.Position := 0.0;
   AxisNuw.Axis[2].Pos26.Speed := 0;
   AxisNuw.Axis[2].Pos26.Reached := FALSE;
   AxisNuw.Axis[2].Pos27.Position := 0.0;
   AxisNuw.Axis[2].Pos27.Speed := 0;
   AxisNuw.Axis[2].Pos27.Reached := FALSE;
   AxisNuw.Axis[2].Pos28.Position := 0.0;
   AxisNuw.Axis[2].Pos28.Speed := 0;
   AxisNuw.Axis[2].Pos28.Reached := FALSE;
   AxisNuw.Axis[2].Pos29.Position := 0.0;
   AxisNuw.Axis[2].Pos29.Speed := 0;
   AxisNuw.Axis[2].Pos29.Reached := FALSE;
   AxisNuw.Axis[2].Pos30.Position := 0.0;
   AxisNuw.Axis[2].Pos30.Speed := 0;
   AxisNuw.Axis[2].Pos30.Reached := FALSE;
   AxisNuw.Axis[3].Pos1.Position := 0.0;
   AxisNuw.Axis[3].Pos1.Speed := 0;
   AxisNuw.Axis[3].Pos1.Reached := FALSE;
   AxisNuw.Axis[3].Pos2.Position := 0.0;
   AxisNuw.Axis[3].Pos2.Speed := 0;
   AxisNuw.Axis[3].Pos2.Reached := FALSE;
   AxisNuw.Axis[3].Pos3.Position := 0.0;
   AxisNuw.Axis[3].Pos3.Speed := 0;
   AxisNuw.Axis[3].Pos3.Reached := FALSE;
   AxisNuw.Axis[3].Pos4.Position := 0.0;
   AxisNuw.Axis[3].Pos4.Speed := 0;
   AxisNuw.Axis[3].Pos4.Reached := FALSE;
   AxisNuw.Axis[3].Pos5.Position := 0.0;
   AxisNuw.Axis[3].Pos5.Speed := 0;
   AxisNuw.Axis[3].Pos5.Reached := FALSE;
   AxisNuw.Axis[3].Pos6.Position := 0.0;
   AxisNuw.Axis[3].Pos6.Speed := 0;
   AxisNuw.Axis[3].Pos6.Reached := FALSE;
   AxisNuw.Axis[3].Pos7.Position := 0.0;
   AxisNuw.Axis[3].Pos7.Speed := 0;
   AxisNuw.Axis[3].Pos7.Reached := FALSE;
   AxisNuw.Axis[3].Pos8.Position := 0.0;
   AxisNuw.Axis[3].Pos8.Speed := 0;
   AxisNuw.Axis[3].Pos8.Reached := FALSE;
   AxisNuw.Axis[3].Pos9.Position := 0.0;
   AxisNuw.Axis[3].Pos9.Speed := 0;
   AxisNuw.Axis[3].Pos9.Reached := FALSE;
   AxisNuw.Axis[3].Pos10.Position := 0.0;
   AxisNuw.Axis[3].Pos10.Speed := 0;
   AxisNuw.Axis[3].Pos10.Reached := FALSE;
   AxisNuw.Axis[3].Pos11.Position := 0.0;
   AxisNuw.Axis[3].Pos11.Speed := 0;
   AxisNuw.Axis[3].Pos11.Reached := FALSE;
   AxisNuw.Axis[3].Pos12.Position := 0.0;
   AxisNuw.Axis[3].Pos12.Speed := 0;
   AxisNuw.Axis[3].Pos12.Reached := FALSE;
   AxisNuw.Axis[3].Pos13.Position := 0.0;
   AxisNuw.Axis[3].Pos13.Speed := 0;
   AxisNuw.Axis[3].Pos13.Reached := FALSE;
   AxisNuw.Axis[3].Pos14.Position := 0.0;
   AxisNuw.Axis[3].Pos14.Speed := 0;
   AxisNuw.Axis[3].Pos14.Reached := FALSE;
   AxisNuw.Axis[3].Pos15.Position := 0.0;
   AxisNuw.Axis[3].Pos15.Speed := 0;
   AxisNuw.Axis[3].Pos15.Reached := FALSE;
   AxisNuw.Axis[3].Pos16.Position := 0.0;
   AxisNuw.Axis[3].Pos16.Speed := 0;
   AxisNuw.Axis[3].Pos16.Reached := FALSE;
   AxisNuw.Axis[3].Pos17.Position := 0.0;
   AxisNuw.Axis[3].Pos17.Speed := 0;
   AxisNuw.Axis[3].Pos17.Reached := FALSE;
   AxisNuw.Axis[3].Pos18.Position := 0.0;
   AxisNuw.Axis[3].Pos18.Speed := 0;
   AxisNuw.Axis[3].Pos18.Reached := FALSE;
   AxisNuw.Axis[3].Pos19.Position := 0.0;
   AxisNuw.Axis[3].Pos19.Speed := 0;
   AxisNuw.Axis[3].Pos19.Reached := FALSE;
   AxisNuw.Axis[3].Pos20.Position := 0.0;
   AxisNuw.Axis[3].Pos20.Speed := 0;
   AxisNuw.Axis[3].Pos20.Reached := FALSE;
   AxisNuw.Axis[3].Pos21.Position := 0.0;
   AxisNuw.Axis[3].Pos21.Speed := 0;
   AxisNuw.Axis[3].Pos21.Reached := FALSE;
   AxisNuw.Axis[3].Pos22.Position := 0.0;
   AxisNuw.Axis[3].Pos22.Speed := 0;
   AxisNuw.Axis[3].Pos22.Reached := FALSE;
   AxisNuw.Axis[3].Pos23.Position := 0.0;
   AxisNuw.Axis[3].Pos23.Speed := 0;
   AxisNuw.Axis[3].Pos23.Reached := FALSE;
   AxisNuw.Axis[3].Pos24.Position := 0.0;
   AxisNuw.Axis[3].Pos24.Speed := 0;
   AxisNuw.Axis[3].Pos24.Reached := FALSE;
   AxisNuw.Axis[3].Pos25.Position := 0.0;
   AxisNuw.Axis[3].Pos25.Speed := 0;
   AxisNuw.Axis[3].Pos25.Reached := FALSE;
   AxisNuw.Axis[3].Pos26.Position := 0.0;
   AxisNuw.Axis[3].Pos26.Speed := 0;
   AxisNuw.Axis[3].Pos26.Reached := FALSE;
   AxisNuw.Axis[3].Pos27.Position := 0.0;
   AxisNuw.Axis[3].Pos27.Speed := 0;
   AxisNuw.Axis[3].Pos27.Reached := FALSE;
   AxisNuw.Axis[3].Pos28.Position := 0.0;
   AxisNuw.Axis[3].Pos28.Speed := 0;
   AxisNuw.Axis[3].Pos28.Reached := FALSE;
   AxisNuw.Axis[3].Pos29.Position := 0.0;
   AxisNuw.Axis[3].Pos29.Speed := 0;
   AxisNuw.Axis[3].Pos29.Reached := FALSE;
   AxisNuw.Axis[3].Pos30.Position := 0.0;
   AxisNuw.Axis[3].Pos30.Speed := 0;
   AxisNuw.Axis[3].Pos30.Reached := FALSE;
   AxisNuw.Axis[4].Pos1.Position := 0.0;
   AxisNuw.Axis[4].Pos1.Speed := 0;
   AxisNuw.Axis[4].Pos1.Reached := FALSE;
   AxisNuw.Axis[4].Pos2.Position := 0.0;
   AxisNuw.Axis[4].Pos2.Speed := 0;
   AxisNuw.Axis[4].Pos2.Reached := FALSE;
   AxisNuw.Axis[4].Pos3.Position := 0.0;
   AxisNuw.Axis[4].Pos3.Speed := 0;
   AxisNuw.Axis[4].Pos3.Reached := FALSE;
   AxisNuw.Axis[4].Pos4.Position := 0.0;
   AxisNuw.Axis[4].Pos4.Speed := 0;
   AxisNuw.Axis[4].Pos4.Reached := FALSE;
   AxisNuw.Axis[4].Pos5.Position := 0.0;
   AxisNuw.Axis[4].Pos5.Speed := 0;
   AxisNuw.Axis[4].Pos5.Reached := FALSE;
   AxisNuw.Axis[4].Pos6.Position := 0.0;
   AxisNuw.Axis[4].Pos6.Speed := 0;
   AxisNuw.Axis[4].Pos6.Reached := FALSE;
   AxisNuw.Axis[4].Pos7.Position := 0.0;
   AxisNuw.Axis[4].Pos7.Speed := 0;
   AxisNuw.Axis[4].Pos7.Reached := FALSE;
   AxisNuw.Axis[4].Pos8.Position := 0.0;
   AxisNuw.Axis[4].Pos8.Speed := 0;
   AxisNuw.Axis[4].Pos8.Reached := FALSE;
   AxisNuw.Axis[4].Pos9.Position := 0.0;
   AxisNuw.Axis[4].Pos9.Speed := 0;
   AxisNuw.Axis[4].Pos9.Reached := FALSE;
   AxisNuw.Axis[4].Pos10.Position := 0.0;
   AxisNuw.Axis[4].Pos10.Speed := 0;
   AxisNuw.Axis[4].Pos10.Reached := FALSE;
   AxisNuw.Axis[4].Pos11.Position := 0.0;
   AxisNuw.Axis[4].Pos11.Speed := 0;
   AxisNuw.Axis[4].Pos11.Reached := FALSE;
   AxisNuw.Axis[4].Pos12.Position := 0.0;
   AxisNuw.Axis[4].Pos12.Speed := 0;
   AxisNuw.Axis[4].Pos12.Reached := FALSE;
   AxisNuw.Axis[4].Pos13.Position := 0.0;
   AxisNuw.Axis[4].Pos13.Speed := 0;
   AxisNuw.Axis[4].Pos13.Reached := FALSE;
   AxisNuw.Axis[4].Pos14.Position := 0.0;
   AxisNuw.Axis[4].Pos14.Speed := 0;
   AxisNuw.Axis[4].Pos14.Reached := FALSE;
   AxisNuw.Axis[4].Pos15.Position := 0.0;
   AxisNuw.Axis[4].Pos15.Speed := 0;
   AxisNuw.Axis[4].Pos15.Reached := FALSE;
   AxisNuw.Axis[4].Pos16.Position := 0.0;
   AxisNuw.Axis[4].Pos16.Speed := 0;
   AxisNuw.Axis[4].Pos16.Reached := FALSE;
   AxisNuw.Axis[4].Pos17.Position := 0.0;
   AxisNuw.Axis[4].Pos17.Speed := 0;
   AxisNuw.Axis[4].Pos17.Reached := FALSE;
   AxisNuw.Axis[4].Pos18.Position := 0.0;
   AxisNuw.Axis[4].Pos18.Speed := 0;
   AxisNuw.Axis[4].Pos18.Reached := FALSE;
   AxisNuw.Axis[4].Pos19.Position := 0.0;
   AxisNuw.Axis[4].Pos19.Speed := 0;
   AxisNuw.Axis[4].Pos19.Reached := FALSE;
   AxisNuw.Axis[4].Pos20.Position := 0.0;
   AxisNuw.Axis[4].Pos20.Speed := 0;
   AxisNuw.Axis[4].Pos20.Reached := FALSE;
   AxisNuw.Axis[4].Pos21.Position := 0.0;
   AxisNuw.Axis[4].Pos21.Speed := 0;
   AxisNuw.Axis[4].Pos21.Reached := FALSE;
   AxisNuw.Axis[4].Pos22.Position := 0.0;
   AxisNuw.Axis[4].Pos22.Speed := 0;
   AxisNuw.Axis[4].Pos22.Reached := FALSE;
   AxisNuw.Axis[4].Pos23.Position := 0.0;
   AxisNuw.Axis[4].Pos23.Speed := 0;
   AxisNuw.Axis[4].Pos23.Reached := FALSE;
   AxisNuw.Axis[4].Pos24.Position := 0.0;
   AxisNuw.Axis[4].Pos24.Speed := 0;
   AxisNuw.Axis[4].Pos24.Reached := FALSE;
   AxisNuw.Axis[4].Pos25.Position := 0.0;
   AxisNuw.Axis[4].Pos25.Speed := 0;
   AxisNuw.Axis[4].Pos25.Reached := FALSE;
   AxisNuw.Axis[4].Pos26.Position := 0.0;
   AxisNuw.Axis[4].Pos26.Speed := 0;
   AxisNuw.Axis[4].Pos26.Reached := FALSE;
   AxisNuw.Axis[4].Pos27.Position := 0.0;
   AxisNuw.Axis[4].Pos27.Speed := 0;
   AxisNuw.Axis[4].Pos27.Reached := FALSE;
   AxisNuw.Axis[4].Pos28.Position := 0.0;
   AxisNuw.Axis[4].Pos28.Speed := 0;
   AxisNuw.Axis[4].Pos28.Reached := FALSE;
   AxisNuw.Axis[4].Pos29.Position := 0.0;
   AxisNuw.Axis[4].Pos29.Speed := 0;
   AxisNuw.Axis[4].Pos29.Reached := FALSE;
   AxisNuw.Axis[4].Pos30.Position := 0.0;
   AxisNuw.Axis[4].Pos30.Speed := 0;
   AxisNuw.Axis[4].Pos30.Reached := FALSE;
   AxisNuw.Axis[5].Pos1.Position := 0.0;
   AxisNuw.Axis[5].Pos1.Speed := 0;
   AxisNuw.Axis[5].Pos1.Reached := FALSE;
   AxisNuw.Axis[5].Pos2.Position := 0.0;
   AxisNuw.Axis[5].Pos2.Speed := 0;
   AxisNuw.Axis[5].Pos2.Reached := FALSE;
   AxisNuw.Axis[5].Pos3.Position := 0.0;
   AxisNuw.Axis[5].Pos3.Speed := 0;
   AxisNuw.Axis[5].Pos3.Reached := FALSE;
   AxisNuw.Axis[5].Pos4.Position := 0.0;
   AxisNuw.Axis[5].Pos4.Speed := 0;
   AxisNuw.Axis[5].Pos4.Reached := FALSE;
   AxisNuw.Axis[5].Pos5.Position := 0.0;
   AxisNuw.Axis[5].Pos5.Speed := 0;
   AxisNuw.Axis[5].Pos5.Reached := FALSE;
   AxisNuw.Axis[5].Pos6.Position := 0.0;
   AxisNuw.Axis[5].Pos6.Speed := 0;
   AxisNuw.Axis[5].Pos6.Reached := FALSE;
   AxisNuw.Axis[5].Pos7.Position := 0.0;
   AxisNuw.Axis[5].Pos7.Speed := 0;
   AxisNuw.Axis[5].Pos7.Reached := FALSE;
   AxisNuw.Axis[5].Pos8.Position := 0.0;
   AxisNuw.Axis[5].Pos8.Speed := 0;
   AxisNuw.Axis[5].Pos8.Reached := FALSE;
   AxisNuw.Axis[5].Pos9.Position := 0.0;
   AxisNuw.Axis[5].Pos9.Speed := 0;
   AxisNuw.Axis[5].Pos9.Reached := FALSE;
   AxisNuw.Axis[5].Pos10.Position := 0.0;
   AxisNuw.Axis[5].Pos10.Speed := 0;
   AxisNuw.Axis[5].Pos10.Reached := FALSE;
   AxisNuw.Axis[5].Pos11.Position := 0.0;
   AxisNuw.Axis[5].Pos11.Speed := 0;
   AxisNuw.Axis[5].Pos11.Reached := FALSE;
   AxisNuw.Axis[5].Pos12.Position := 0.0;
   AxisNuw.Axis[5].Pos12.Speed := 0;
   AxisNuw.Axis[5].Pos12.Reached := FALSE;
   AxisNuw.Axis[5].Pos13.Position := 0.0;
   AxisNuw.Axis[5].Pos13.Speed := 0;
   AxisNuw.Axis[5].Pos13.Reached := FALSE;
   AxisNuw.Axis[5].Pos14.Position := 0.0;
   AxisNuw.Axis[5].Pos14.Speed := 0;
   AxisNuw.Axis[5].Pos14.Reached := FALSE;
   AxisNuw.Axis[5].Pos15.Position := 0.0;
   AxisNuw.Axis[5].Pos15.Speed := 0;
   AxisNuw.Axis[5].Pos15.Reached := FALSE;
   AxisNuw.Axis[5].Pos16.Position := 0.0;
   AxisNuw.Axis[5].Pos16.Speed := 0;
   AxisNuw.Axis[5].Pos16.Reached := FALSE;
   AxisNuw.Axis[5].Pos17.Position := 0.0;
   AxisNuw.Axis[5].Pos17.Speed := 0;
   AxisNuw.Axis[5].Pos17.Reached := FALSE;
   AxisNuw.Axis[5].Pos18.Position := 0.0;
   AxisNuw.Axis[5].Pos18.Speed := 0;
   AxisNuw.Axis[5].Pos18.Reached := FALSE;
   AxisNuw.Axis[5].Pos19.Position := 0.0;
   AxisNuw.Axis[5].Pos19.Speed := 0;
   AxisNuw.Axis[5].Pos19.Reached := FALSE;
   AxisNuw.Axis[5].Pos20.Position := 0.0;
   AxisNuw.Axis[5].Pos20.Speed := 0;
   AxisNuw.Axis[5].Pos20.Reached := FALSE;
   AxisNuw.Axis[5].Pos21.Position := 0.0;
   AxisNuw.Axis[5].Pos21.Speed := 0;
   AxisNuw.Axis[5].Pos21.Reached := FALSE;
   AxisNuw.Axis[5].Pos22.Position := 0.0;
   AxisNuw.Axis[5].Pos22.Speed := 0;
   AxisNuw.Axis[5].Pos22.Reached := FALSE;
   AxisNuw.Axis[5].Pos23.Position := 0.0;
   AxisNuw.Axis[5].Pos23.Speed := 0;
   AxisNuw.Axis[5].Pos23.Reached := FALSE;
   AxisNuw.Axis[5].Pos24.Position := 0.0;
   AxisNuw.Axis[5].Pos24.Speed := 0;
   AxisNuw.Axis[5].Pos24.Reached := FALSE;
   AxisNuw.Axis[5].Pos25.Position := 0.0;
   AxisNuw.Axis[5].Pos25.Speed := 0;
   AxisNuw.Axis[5].Pos25.Reached := FALSE;
   AxisNuw.Axis[5].Pos26.Position := 0.0;
   AxisNuw.Axis[5].Pos26.Speed := 0;
   AxisNuw.Axis[5].Pos26.Reached := FALSE;
   AxisNuw.Axis[5].Pos27.Position := 0.0;
   AxisNuw.Axis[5].Pos27.Speed := 0;
   AxisNuw.Axis[5].Pos27.Reached := FALSE;
   AxisNuw.Axis[5].Pos28.Position := 0.0;
   AxisNuw.Axis[5].Pos28.Speed := 0;
   AxisNuw.Axis[5].Pos28.Reached := FALSE;
   AxisNuw.Axis[5].Pos29.Position := 0.0;
   AxisNuw.Axis[5].Pos29.Speed := 0;
   AxisNuw.Axis[5].Pos29.Reached := FALSE;
   AxisNuw.Axis[5].Pos30.Position := 0.0;
   AxisNuw.Axis[5].Pos30.Speed := 0;
   AxisNuw.Axis[5].Pos30.Reached := FALSE;
   AxisNuw.Axis[6].Pos1.Position := 0.0;
   AxisNuw.Axis[6].Pos1.Speed := 0;
   AxisNuw.Axis[6].Pos1.Reached := FALSE;
   AxisNuw.Axis[6].Pos2.Position := 0.0;
   AxisNuw.Axis[6].Pos2.Speed := 0;
   AxisNuw.Axis[6].Pos2.Reached := FALSE;
   AxisNuw.Axis[6].Pos3.Position := 0.0;
   AxisNuw.Axis[6].Pos3.Speed := 0;
   AxisNuw.Axis[6].Pos3.Reached := FALSE;
   AxisNuw.Axis[6].Pos4.Position := 0.0;
   AxisNuw.Axis[6].Pos4.Speed := 0;
   AxisNuw.Axis[6].Pos4.Reached := FALSE;
   AxisNuw.Axis[6].Pos5.Position := 0.0;
   AxisNuw.Axis[6].Pos5.Speed := 0;
   AxisNuw.Axis[6].Pos5.Reached := FALSE;
   AxisNuw.Axis[6].Pos6.Position := 0.0;
   AxisNuw.Axis[6].Pos6.Speed := 0;
   AxisNuw.Axis[6].Pos6.Reached := FALSE;
   AxisNuw.Axis[6].Pos7.Position := 0.0;
   AxisNuw.Axis[6].Pos7.Speed := 0;
   AxisNuw.Axis[6].Pos7.Reached := FALSE;
   AxisNuw.Axis[6].Pos8.Position := 0.0;
   AxisNuw.Axis[6].Pos8.Speed := 0;
   AxisNuw.Axis[6].Pos8.Reached := FALSE;
   AxisNuw.Axis[6].Pos9.Position := 0.0;
   AxisNuw.Axis[6].Pos9.Speed := 0;
   AxisNuw.Axis[6].Pos9.Reached := FALSE;
   AxisNuw.Axis[6].Pos10.Position := 0.0;
   AxisNuw.Axis[6].Pos10.Speed := 0;
   AxisNuw.Axis[6].Pos10.Reached := FALSE;
   AxisNuw.Axis[6].Pos11.Position := 0.0;
   AxisNuw.Axis[6].Pos11.Speed := 0;
   AxisNuw.Axis[6].Pos11.Reached := FALSE;
   AxisNuw.Axis[6].Pos12.Position := 0.0;
   AxisNuw.Axis[6].Pos12.Speed := 0;
   AxisNuw.Axis[6].Pos12.Reached := FALSE;
   AxisNuw.Axis[6].Pos13.Position := 0.0;
   AxisNuw.Axis[6].Pos13.Speed := 0;
   AxisNuw.Axis[6].Pos13.Reached := FALSE;
   AxisNuw.Axis[6].Pos14.Position := 0.0;
   AxisNuw.Axis[6].Pos14.Speed := 0;
   AxisNuw.Axis[6].Pos14.Reached := FALSE;
   AxisNuw.Axis[6].Pos15.Position := 0.0;
   AxisNuw.Axis[6].Pos15.Speed := 0;
   AxisNuw.Axis[6].Pos15.Reached := FALSE;
   AxisNuw.Axis[6].Pos16.Position := 0.0;
   AxisNuw.Axis[6].Pos16.Speed := 0;
   AxisNuw.Axis[6].Pos16.Reached := FALSE;
   AxisNuw.Axis[6].Pos17.Position := 0.0;
   AxisNuw.Axis[6].Pos17.Speed := 0;
   AxisNuw.Axis[6].Pos17.Reached := FALSE;
   AxisNuw.Axis[6].Pos18.Position := 0.0;
   AxisNuw.Axis[6].Pos18.Speed := 0;
   AxisNuw.Axis[6].Pos18.Reached := FALSE;
   AxisNuw.Axis[6].Pos19.Position := 0.0;
   AxisNuw.Axis[6].Pos19.Speed := 0;
   AxisNuw.Axis[6].Pos19.Reached := FALSE;
   AxisNuw.Axis[6].Pos20.Position := 0.0;
   AxisNuw.Axis[6].Pos20.Speed := 0;
   AxisNuw.Axis[6].Pos20.Reached := FALSE;
   AxisNuw.Axis[6].Pos21.Position := 0.0;
   AxisNuw.Axis[6].Pos21.Speed := 0;
   AxisNuw.Axis[6].Pos21.Reached := FALSE;
   AxisNuw.Axis[6].Pos22.Position := 0.0;
   AxisNuw.Axis[6].Pos22.Speed := 0;
   AxisNuw.Axis[6].Pos22.Reached := FALSE;
   AxisNuw.Axis[6].Pos23.Position := 0.0;
   AxisNuw.Axis[6].Pos23.Speed := 0;
   AxisNuw.Axis[6].Pos23.Reached := FALSE;
   AxisNuw.Axis[6].Pos24.Position := 0.0;
   AxisNuw.Axis[6].Pos24.Speed := 0;
   AxisNuw.Axis[6].Pos24.Reached := FALSE;
   AxisNuw.Axis[6].Pos25.Position := 0.0;
   AxisNuw.Axis[6].Pos25.Speed := 0;
   AxisNuw.Axis[6].Pos25.Reached := FALSE;
   AxisNuw.Axis[6].Pos26.Position := 0.0;
   AxisNuw.Axis[6].Pos26.Speed := 0;
   AxisNuw.Axis[6].Pos26.Reached := FALSE;
   AxisNuw.Axis[6].Pos27.Position := 0.0;
   AxisNuw.Axis[6].Pos27.Speed := 0;
   AxisNuw.Axis[6].Pos27.Reached := FALSE;
   AxisNuw.Axis[6].Pos28.Position := 0.0;
   AxisNuw.Axis[6].Pos28.Speed := 0;
   AxisNuw.Axis[6].Pos28.Reached := FALSE;
   AxisNuw.Axis[6].Pos29.Position := 0.0;
   AxisNuw.Axis[6].Pos29.Speed := 0;
   AxisNuw.Axis[6].Pos29.Reached := FALSE;
   AxisNuw.Axis[6].Pos30.Position := 0.0;
   AxisNuw.Axis[6].Pos30.Speed := 0;
   AxisNuw.Axis[6].Pos30.Reached := FALSE;
   AxisNuw.Axis[7].Pos1.Position := 0.0;
   AxisNuw.Axis[7].Pos1.Speed := 0;
   AxisNuw.Axis[7].Pos1.Reached := FALSE;
   AxisNuw.Axis[7].Pos2.Position := 0.0;
   AxisNuw.Axis[7].Pos2.Speed := 0;
   AxisNuw.Axis[7].Pos2.Reached := FALSE;
   AxisNuw.Axis[7].Pos3.Position := 0.0;
   AxisNuw.Axis[7].Pos3.Speed := 0;
   AxisNuw.Axis[7].Pos3.Reached := FALSE;
   AxisNuw.Axis[7].Pos4.Position := 0.0;
   AxisNuw.Axis[7].Pos4.Speed := 0;
   AxisNuw.Axis[7].Pos4.Reached := FALSE;
   AxisNuw.Axis[7].Pos5.Position := 0.0;
   AxisNuw.Axis[7].Pos5.Speed := 0;
   AxisNuw.Axis[7].Pos5.Reached := FALSE;
   AxisNuw.Axis[7].Pos6.Position := 0.0;
   AxisNuw.Axis[7].Pos6.Speed := 0;
   AxisNuw.Axis[7].Pos6.Reached := FALSE;
   AxisNuw.Axis[7].Pos7.Position := 0.0;
   AxisNuw.Axis[7].Pos7.Speed := 0;
   AxisNuw.Axis[7].Pos7.Reached := FALSE;
   AxisNuw.Axis[7].Pos8.Position := 0.0;
   AxisNuw.Axis[7].Pos8.Speed := 0;
   AxisNuw.Axis[7].Pos8.Reached := FALSE;
   AxisNuw.Axis[7].Pos9.Position := 0.0;
   AxisNuw.Axis[7].Pos9.Speed := 0;
   AxisNuw.Axis[7].Pos9.Reached := FALSE;
   AxisNuw.Axis[7].Pos10.Position := 0.0;
   AxisNuw.Axis[7].Pos10.Speed := 0;
   AxisNuw.Axis[7].Pos10.Reached := FALSE;
   AxisNuw.Axis[7].Pos11.Position := 0.0;
   AxisNuw.Axis[7].Pos11.Speed := 0;
   AxisNuw.Axis[7].Pos11.Reached := FALSE;
   AxisNuw.Axis[7].Pos12.Position := 0.0;
   AxisNuw.Axis[7].Pos12.Speed := 0;
   AxisNuw.Axis[7].Pos12.Reached := FALSE;
   AxisNuw.Axis[7].Pos13.Position := 0.0;
   AxisNuw.Axis[7].Pos13.Speed := 0;
   AxisNuw.Axis[7].Pos13.Reached := FALSE;
   AxisNuw.Axis[7].Pos14.Position := 0.0;
   AxisNuw.Axis[7].Pos14.Speed := 0;
   AxisNuw.Axis[7].Pos14.Reached := FALSE;
   AxisNuw.Axis[7].Pos15.Position := 0.0;
   AxisNuw.Axis[7].Pos15.Speed := 0;
   AxisNuw.Axis[7].Pos15.Reached := FALSE;
   AxisNuw.Axis[7].Pos16.Position := 0.0;
   AxisNuw.Axis[7].Pos16.Speed := 0;
   AxisNuw.Axis[7].Pos16.Reached := FALSE;
   AxisNuw.Axis[7].Pos17.Position := 0.0;
   AxisNuw.Axis[7].Pos17.Speed := 0;
   AxisNuw.Axis[7].Pos17.Reached := FALSE;
   AxisNuw.Axis[7].Pos18.Position := 0.0;
   AxisNuw.Axis[7].Pos18.Speed := 0;
   AxisNuw.Axis[7].Pos18.Reached := FALSE;
   AxisNuw.Axis[7].Pos19.Position := 0.0;
   AxisNuw.Axis[7].Pos19.Speed := 0;
   AxisNuw.Axis[7].Pos19.Reached := FALSE;
   AxisNuw.Axis[7].Pos20.Position := 0.0;
   AxisNuw.Axis[7].Pos20.Speed := 0;
   AxisNuw.Axis[7].Pos20.Reached := FALSE;
   AxisNuw.Axis[7].Pos21.Position := 0.0;
   AxisNuw.Axis[7].Pos21.Speed := 0;
   AxisNuw.Axis[7].Pos21.Reached := FALSE;
   AxisNuw.Axis[7].Pos22.Position := 0.0;
   AxisNuw.Axis[7].Pos22.Speed := 0;
   AxisNuw.Axis[7].Pos22.Reached := FALSE;
   AxisNuw.Axis[7].Pos23.Position := 0.0;
   AxisNuw.Axis[7].Pos23.Speed := 0;
   AxisNuw.Axis[7].Pos23.Reached := FALSE;
   AxisNuw.Axis[7].Pos24.Position := 0.0;
   AxisNuw.Axis[7].Pos24.Speed := 0;
   AxisNuw.Axis[7].Pos24.Reached := FALSE;
   AxisNuw.Axis[7].Pos25.Position := 0.0;
   AxisNuw.Axis[7].Pos25.Speed := 0;
   AxisNuw.Axis[7].Pos25.Reached := FALSE;
   AxisNuw.Axis[7].Pos26.Position := 0.0;
   AxisNuw.Axis[7].Pos26.Speed := 0;
   AxisNuw.Axis[7].Pos26.Reached := FALSE;
   AxisNuw.Axis[7].Pos27.Position := 0.0;
   AxisNuw.Axis[7].Pos27.Speed := 0;
   AxisNuw.Axis[7].Pos27.Reached := FALSE;
   AxisNuw.Axis[7].Pos28.Position := 0.0;
   AxisNuw.Axis[7].Pos28.Speed := 0;
   AxisNuw.Axis[7].Pos28.Reached := FALSE;
   AxisNuw.Axis[7].Pos29.Position := 0.0;
   AxisNuw.Axis[7].Pos29.Speed := 0;
   AxisNuw.Axis[7].Pos29.Reached := FALSE;
   AxisNuw.Axis[7].Pos30.Position := 0.0;
   AxisNuw.Axis[7].Pos30.Speed := 0;
   AxisNuw.Axis[7].Pos30.Reached := FALSE;
   AxisNuw.Axis[8].Pos1.Position := 0.0;
   AxisNuw.Axis[8].Pos1.Speed := 0;
   AxisNuw.Axis[8].Pos1.Reached := FALSE;
   AxisNuw.Axis[8].Pos2.Position := 0.0;
   AxisNuw.Axis[8].Pos2.Speed := 0;
   AxisNuw.Axis[8].Pos2.Reached := FALSE;
   AxisNuw.Axis[8].Pos3.Position := 0.0;
   AxisNuw.Axis[8].Pos3.Speed := 0;
   AxisNuw.Axis[8].Pos3.Reached := FALSE;
   AxisNuw.Axis[8].Pos4.Position := 0.0;
   AxisNuw.Axis[8].Pos4.Speed := 0;
   AxisNuw.Axis[8].Pos4.Reached := FALSE;
   AxisNuw.Axis[8].Pos5.Position := 0.0;
   AxisNuw.Axis[8].Pos5.Speed := 0;
   AxisNuw.Axis[8].Pos5.Reached := FALSE;
   AxisNuw.Axis[8].Pos6.Position := 0.0;
   AxisNuw.Axis[8].Pos6.Speed := 0;
   AxisNuw.Axis[8].Pos6.Reached := FALSE;
   AxisNuw.Axis[8].Pos7.Position := 0.0;
   AxisNuw.Axis[8].Pos7.Speed := 0;
   AxisNuw.Axis[8].Pos7.Reached := FALSE;
   AxisNuw.Axis[8].Pos8.Position := 0.0;
   AxisNuw.Axis[8].Pos8.Speed := 0;
   AxisNuw.Axis[8].Pos8.Reached := FALSE;
   AxisNuw.Axis[8].Pos9.Position := 0.0;
   AxisNuw.Axis[8].Pos9.Speed := 0;
   AxisNuw.Axis[8].Pos9.Reached := FALSE;
   AxisNuw.Axis[8].Pos10.Position := 0.0;
   AxisNuw.Axis[8].Pos10.Speed := 0;
   AxisNuw.Axis[8].Pos10.Reached := FALSE;
   AxisNuw.Axis[8].Pos11.Position := 0.0;
   AxisNuw.Axis[8].Pos11.Speed := 0;
   AxisNuw.Axis[8].Pos11.Reached := FALSE;
   AxisNuw.Axis[8].Pos12.Position := 0.0;
   AxisNuw.Axis[8].Pos12.Speed := 0;
   AxisNuw.Axis[8].Pos12.Reached := FALSE;
   AxisNuw.Axis[8].Pos13.Position := 0.0;
   AxisNuw.Axis[8].Pos13.Speed := 0;
   AxisNuw.Axis[8].Pos13.Reached := FALSE;
   AxisNuw.Axis[8].Pos14.Position := 0.0;
   AxisNuw.Axis[8].Pos14.Speed := 0;
   AxisNuw.Axis[8].Pos14.Reached := FALSE;
   AxisNuw.Axis[8].Pos15.Position := 0.0;
   AxisNuw.Axis[8].Pos15.Speed := 0;
   AxisNuw.Axis[8].Pos15.Reached := FALSE;
   AxisNuw.Axis[8].Pos16.Position := 0.0;
   AxisNuw.Axis[8].Pos16.Speed := 0;
   AxisNuw.Axis[8].Pos16.Reached := FALSE;
   AxisNuw.Axis[8].Pos17.Position := 0.0;
   AxisNuw.Axis[8].Pos17.Speed := 0;
   AxisNuw.Axis[8].Pos17.Reached := FALSE;
   AxisNuw.Axis[8].Pos18.Position := 0.0;
   AxisNuw.Axis[8].Pos18.Speed := 0;
   AxisNuw.Axis[8].Pos18.Reached := FALSE;
   AxisNuw.Axis[8].Pos19.Position := 0.0;
   AxisNuw.Axis[8].Pos19.Speed := 0;
   AxisNuw.Axis[8].Pos19.Reached := FALSE;
   AxisNuw.Axis[8].Pos20.Position := 0.0;
   AxisNuw.Axis[8].Pos20.Speed := 0;
   AxisNuw.Axis[8].Pos20.Reached := FALSE;
   AxisNuw.Axis[8].Pos21.Position := 0.0;
   AxisNuw.Axis[8].Pos21.Speed := 0;
   AxisNuw.Axis[8].Pos21.Reached := FALSE;
   AxisNuw.Axis[8].Pos22.Position := 0.0;
   AxisNuw.Axis[8].Pos22.Speed := 0;
   AxisNuw.Axis[8].Pos22.Reached := FALSE;
   AxisNuw.Axis[8].Pos23.Position := 0.0;
   AxisNuw.Axis[8].Pos23.Speed := 0;
   AxisNuw.Axis[8].Pos23.Reached := FALSE;
   AxisNuw.Axis[8].Pos24.Position := 0.0;
   AxisNuw.Axis[8].Pos24.Speed := 0;
   AxisNuw.Axis[8].Pos24.Reached := FALSE;
   AxisNuw.Axis[8].Pos25.Position := 0.0;
   AxisNuw.Axis[8].Pos25.Speed := 0;
   AxisNuw.Axis[8].Pos25.Reached := FALSE;
   AxisNuw.Axis[8].Pos26.Position := 0.0;
   AxisNuw.Axis[8].Pos26.Speed := 0;
   AxisNuw.Axis[8].Pos26.Reached := FALSE;
   AxisNuw.Axis[8].Pos27.Position := 0.0;
   AxisNuw.Axis[8].Pos27.Speed := 0;
   AxisNuw.Axis[8].Pos27.Reached := FALSE;
   AxisNuw.Axis[8].Pos28.Position := 0.0;
   AxisNuw.Axis[8].Pos28.Speed := 0;
   AxisNuw.Axis[8].Pos28.Reached := FALSE;
   AxisNuw.Axis[8].Pos29.Position := 0.0;
   AxisNuw.Axis[8].Pos29.Speed := 0;
   AxisNuw.Axis[8].Pos29.Reached := FALSE;
   AxisNuw.Axis[8].Pos30.Position := 0.0;
   AxisNuw.Axis[8].Pos30.Speed := 0;
   AxisNuw.Axis[8].Pos30.Reached := FALSE;
   AxisNuw.Axis[9].Pos1.Position := 0.0;
   AxisNuw.Axis[9].Pos1.Speed := 0;
   AxisNuw.Axis[9].Pos1.Reached := FALSE;
   AxisNuw.Axis[9].Pos2.Position := 0.0;
   AxisNuw.Axis[9].Pos2.Speed := 0;
   AxisNuw.Axis[9].Pos2.Reached := FALSE;
   AxisNuw.Axis[9].Pos3.Position := 0.0;
   AxisNuw.Axis[9].Pos3.Speed := 0;
   AxisNuw.Axis[9].Pos3.Reached := FALSE;
   AxisNuw.Axis[9].Pos4.Position := 0.0;
   AxisNuw.Axis[9].Pos4.Speed := 0;
   AxisNuw.Axis[9].Pos4.Reached := FALSE;
   AxisNuw.Axis[9].Pos5.Position := 0.0;
   AxisNuw.Axis[9].Pos5.Speed := 0;
   AxisNuw.Axis[9].Pos5.Reached := FALSE;
   AxisNuw.Axis[9].Pos6.Position := 0.0;
   AxisNuw.Axis[9].Pos6.Speed := 0;
   AxisNuw.Axis[9].Pos6.Reached := FALSE;
   AxisNuw.Axis[9].Pos7.Position := 0.0;
   AxisNuw.Axis[9].Pos7.Speed := 0;
   AxisNuw.Axis[9].Pos7.Reached := FALSE;
   AxisNuw.Axis[9].Pos8.Position := 0.0;
   AxisNuw.Axis[9].Pos8.Speed := 0;
   AxisNuw.Axis[9].Pos8.Reached := FALSE;
   AxisNuw.Axis[9].Pos9.Position := 0.0;
   AxisNuw.Axis[9].Pos9.Speed := 0;
   AxisNuw.Axis[9].Pos9.Reached := FALSE;
   AxisNuw.Axis[9].Pos10.Position := 0.0;
   AxisNuw.Axis[9].Pos10.Speed := 0;
   AxisNuw.Axis[9].Pos10.Reached := FALSE;
   AxisNuw.Axis[9].Pos11.Position := 0.0;
   AxisNuw.Axis[9].Pos11.Speed := 0;
   AxisNuw.Axis[9].Pos11.Reached := FALSE;
   AxisNuw.Axis[9].Pos12.Position := 0.0;
   AxisNuw.Axis[9].Pos12.Speed := 0;
   AxisNuw.Axis[9].Pos12.Reached := FALSE;
   AxisNuw.Axis[9].Pos13.Position := 0.0;
   AxisNuw.Axis[9].Pos13.Speed := 0;
   AxisNuw.Axis[9].Pos13.Reached := FALSE;
   AxisNuw.Axis[9].Pos14.Position := 0.0;
   AxisNuw.Axis[9].Pos14.Speed := 0;
   AxisNuw.Axis[9].Pos14.Reached := FALSE;
   AxisNuw.Axis[9].Pos15.Position := 0.0;
   AxisNuw.Axis[9].Pos15.Speed := 0;
   AxisNuw.Axis[9].Pos15.Reached := FALSE;
   AxisNuw.Axis[9].Pos16.Position := 0.0;
   AxisNuw.Axis[9].Pos16.Speed := 0;
   AxisNuw.Axis[9].Pos16.Reached := FALSE;
   AxisNuw.Axis[9].Pos17.Position := 0.0;
   AxisNuw.Axis[9].Pos17.Speed := 0;
   AxisNuw.Axis[9].Pos17.Reached := FALSE;
   AxisNuw.Axis[9].Pos18.Position := 0.0;
   AxisNuw.Axis[9].Pos18.Speed := 0;
   AxisNuw.Axis[9].Pos18.Reached := FALSE;
   AxisNuw.Axis[9].Pos19.Position := 0.0;
   AxisNuw.Axis[9].Pos19.Speed := 0;
   AxisNuw.Axis[9].Pos19.Reached := FALSE;
   AxisNuw.Axis[9].Pos20.Position := 0.0;
   AxisNuw.Axis[9].Pos20.Speed := 0;
   AxisNuw.Axis[9].Pos20.Reached := FALSE;
   AxisNuw.Axis[9].Pos21.Position := 0.0;
   AxisNuw.Axis[9].Pos21.Speed := 0;
   AxisNuw.Axis[9].Pos21.Reached := FALSE;
   AxisNuw.Axis[9].Pos22.Position := 0.0;
   AxisNuw.Axis[9].Pos22.Speed := 0;
   AxisNuw.Axis[9].Pos22.Reached := FALSE;
   AxisNuw.Axis[9].Pos23.Position := 0.0;
   AxisNuw.Axis[9].Pos23.Speed := 0;
   AxisNuw.Axis[9].Pos23.Reached := FALSE;
   AxisNuw.Axis[9].Pos24.Position := 0.0;
   AxisNuw.Axis[9].Pos24.Speed := 0;
   AxisNuw.Axis[9].Pos24.Reached := FALSE;
   AxisNuw.Axis[9].Pos25.Position := 0.0;
   AxisNuw.Axis[9].Pos25.Speed := 0;
   AxisNuw.Axis[9].Pos25.Reached := FALSE;
   AxisNuw.Axis[9].Pos26.Position := 0.0;
   AxisNuw.Axis[9].Pos26.Speed := 0;
   AxisNuw.Axis[9].Pos26.Reached := FALSE;
   AxisNuw.Axis[9].Pos27.Position := 0.0;
   AxisNuw.Axis[9].Pos27.Speed := 0;
   AxisNuw.Axis[9].Pos27.Reached := FALSE;
   AxisNuw.Axis[9].Pos28.Position := 0.0;
   AxisNuw.Axis[9].Pos28.Speed := 0;
   AxisNuw.Axis[9].Pos28.Reached := FALSE;
   AxisNuw.Axis[9].Pos29.Position := 0.0;
   AxisNuw.Axis[9].Pos29.Speed := 0;
   AxisNuw.Axis[9].Pos29.Reached := FALSE;
   AxisNuw.Axis[9].Pos30.Position := 0.0;
   AxisNuw.Axis[9].Pos30.Speed := 0;
   AxisNuw.Axis[9].Pos30.Reached := FALSE;
   AxisNuw.Axis[10].Pos1.Position := 0.0;
   AxisNuw.Axis[10].Pos1.Speed := 0;
   AxisNuw.Axis[10].Pos1.Reached := FALSE;
   AxisNuw.Axis[10].Pos2.Position := 0.0;
   AxisNuw.Axis[10].Pos2.Speed := 0;
   AxisNuw.Axis[10].Pos2.Reached := FALSE;
   AxisNuw.Axis[10].Pos3.Position := 0.0;
   AxisNuw.Axis[10].Pos3.Speed := 0;
   AxisNuw.Axis[10].Pos3.Reached := FALSE;
   AxisNuw.Axis[10].Pos4.Position := 0.0;
   AxisNuw.Axis[10].Pos4.Speed := 0;
   AxisNuw.Axis[10].Pos4.Reached := FALSE;
   AxisNuw.Axis[10].Pos5.Position := 0.0;
   AxisNuw.Axis[10].Pos5.Speed := 0;
   AxisNuw.Axis[10].Pos5.Reached := FALSE;
   AxisNuw.Axis[10].Pos6.Position := 0.0;
   AxisNuw.Axis[10].Pos6.Speed := 0;
   AxisNuw.Axis[10].Pos6.Reached := FALSE;
   AxisNuw.Axis[10].Pos7.Position := 0.0;
   AxisNuw.Axis[10].Pos7.Speed := 0;
   AxisNuw.Axis[10].Pos7.Reached := FALSE;
   AxisNuw.Axis[10].Pos8.Position := 0.0;
   AxisNuw.Axis[10].Pos8.Speed := 0;
   AxisNuw.Axis[10].Pos8.Reached := FALSE;
   AxisNuw.Axis[10].Pos9.Position := 0.0;
   AxisNuw.Axis[10].Pos9.Speed := 0;
   AxisNuw.Axis[10].Pos9.Reached := FALSE;
   AxisNuw.Axis[10].Pos10.Position := 0.0;
   AxisNuw.Axis[10].Pos10.Speed := 0;
   AxisNuw.Axis[10].Pos10.Reached := FALSE;
   AxisNuw.Axis[10].Pos11.Position := 0.0;
   AxisNuw.Axis[10].Pos11.Speed := 0;
   AxisNuw.Axis[10].Pos11.Reached := FALSE;
   AxisNuw.Axis[10].Pos12.Position := 0.0;
   AxisNuw.Axis[10].Pos12.Speed := 0;
   AxisNuw.Axis[10].Pos12.Reached := FALSE;
   AxisNuw.Axis[10].Pos13.Position := 0.0;
   AxisNuw.Axis[10].Pos13.Speed := 0;
   AxisNuw.Axis[10].Pos13.Reached := FALSE;
   AxisNuw.Axis[10].Pos14.Position := 0.0;
   AxisNuw.Axis[10].Pos14.Speed := 0;
   AxisNuw.Axis[10].Pos14.Reached := FALSE;
   AxisNuw.Axis[10].Pos15.Position := 0.0;
   AxisNuw.Axis[10].Pos15.Speed := 0;
   AxisNuw.Axis[10].Pos15.Reached := FALSE;
   AxisNuw.Axis[10].Pos16.Position := 0.0;
   AxisNuw.Axis[10].Pos16.Speed := 0;
   AxisNuw.Axis[10].Pos16.Reached := FALSE;
   AxisNuw.Axis[10].Pos17.Position := 0.0;
   AxisNuw.Axis[10].Pos17.Speed := 0;
   AxisNuw.Axis[10].Pos17.Reached := FALSE;
   AxisNuw.Axis[10].Pos18.Position := 0.0;
   AxisNuw.Axis[10].Pos18.Speed := 0;
   AxisNuw.Axis[10].Pos18.Reached := FALSE;
   AxisNuw.Axis[10].Pos19.Position := 0.0;
   AxisNuw.Axis[10].Pos19.Speed := 0;
   AxisNuw.Axis[10].Pos19.Reached := FALSE;
   AxisNuw.Axis[10].Pos20.Position := 0.0;
   AxisNuw.Axis[10].Pos20.Speed := 0;
   AxisNuw.Axis[10].Pos20.Reached := FALSE;
   AxisNuw.Axis[10].Pos21.Position := 0.0;
   AxisNuw.Axis[10].Pos21.Speed := 0;
   AxisNuw.Axis[10].Pos21.Reached := FALSE;
   AxisNuw.Axis[10].Pos22.Position := 0.0;
   AxisNuw.Axis[10].Pos22.Speed := 0;
   AxisNuw.Axis[10].Pos22.Reached := FALSE;
   AxisNuw.Axis[10].Pos23.Position := 0.0;
   AxisNuw.Axis[10].Pos23.Speed := 0;
   AxisNuw.Axis[10].Pos23.Reached := FALSE;
   AxisNuw.Axis[10].Pos24.Position := 0.0;
   AxisNuw.Axis[10].Pos24.Speed := 0;
   AxisNuw.Axis[10].Pos24.Reached := FALSE;
   AxisNuw.Axis[10].Pos25.Position := 0.0;
   AxisNuw.Axis[10].Pos25.Speed := 0;
   AxisNuw.Axis[10].Pos25.Reached := FALSE;
   AxisNuw.Axis[10].Pos26.Position := 0.0;
   AxisNuw.Axis[10].Pos26.Speed := 0;
   AxisNuw.Axis[10].Pos26.Reached := FALSE;
   AxisNuw.Axis[10].Pos27.Position := 0.0;
   AxisNuw.Axis[10].Pos27.Speed := 0;
   AxisNuw.Axis[10].Pos27.Reached := FALSE;
   AxisNuw.Axis[10].Pos28.Position := 0.0;
   AxisNuw.Axis[10].Pos28.Speed := 0;
   AxisNuw.Axis[10].Pos28.Reached := FALSE;
   AxisNuw.Axis[10].Pos29.Position := 0.0;
   AxisNuw.Axis[10].Pos29.Speed := 0;
   AxisNuw.Axis[10].Pos29.Reached := FALSE;
   AxisNuw.Axis[10].Pos30.Position := 0.0;
   AxisNuw.Axis[10].Pos30.Speed := 0;
   AxisNuw.Axis[10].Pos30.Reached := FALSE;
   AxisNuw.Axis[11].Pos1.Position := 0.0;
   AxisNuw.Axis[11].Pos1.Speed := 0;
   AxisNuw.Axis[11].Pos1.Reached := FALSE;
   AxisNuw.Axis[11].Pos2.Position := 0.0;
   AxisNuw.Axis[11].Pos2.Speed := 0;
   AxisNuw.Axis[11].Pos2.Reached := FALSE;
   AxisNuw.Axis[11].Pos3.Position := 0.0;
   AxisNuw.Axis[11].Pos3.Speed := 0;
   AxisNuw.Axis[11].Pos3.Reached := FALSE;
   AxisNuw.Axis[11].Pos4.Position := 0.0;
   AxisNuw.Axis[11].Pos4.Speed := 0;
   AxisNuw.Axis[11].Pos4.Reached := FALSE;
   AxisNuw.Axis[11].Pos5.Position := 0.0;
   AxisNuw.Axis[11].Pos5.Speed := 0;
   AxisNuw.Axis[11].Pos5.Reached := FALSE;
   AxisNuw.Axis[11].Pos6.Position := 0.0;
   AxisNuw.Axis[11].Pos6.Speed := 0;
   AxisNuw.Axis[11].Pos6.Reached := FALSE;
   AxisNuw.Axis[11].Pos7.Position := 0.0;
   AxisNuw.Axis[11].Pos7.Speed := 0;
   AxisNuw.Axis[11].Pos7.Reached := FALSE;
   AxisNuw.Axis[11].Pos8.Position := 0.0;
   AxisNuw.Axis[11].Pos8.Speed := 0;
   AxisNuw.Axis[11].Pos8.Reached := FALSE;
   AxisNuw.Axis[11].Pos9.Position := 0.0;
   AxisNuw.Axis[11].Pos9.Speed := 0;
   AxisNuw.Axis[11].Pos9.Reached := FALSE;
   AxisNuw.Axis[11].Pos10.Position := 0.0;
   AxisNuw.Axis[11].Pos10.Speed := 0;
   AxisNuw.Axis[11].Pos10.Reached := FALSE;
   AxisNuw.Axis[11].Pos11.Position := 0.0;
   AxisNuw.Axis[11].Pos11.Speed := 0;
   AxisNuw.Axis[11].Pos11.Reached := FALSE;
   AxisNuw.Axis[11].Pos12.Position := 0.0;
   AxisNuw.Axis[11].Pos12.Speed := 0;
   AxisNuw.Axis[11].Pos12.Reached := FALSE;
   AxisNuw.Axis[11].Pos13.Position := 0.0;
   AxisNuw.Axis[11].Pos13.Speed := 0;
   AxisNuw.Axis[11].Pos13.Reached := FALSE;
   AxisNuw.Axis[11].Pos14.Position := 0.0;
   AxisNuw.Axis[11].Pos14.Speed := 0;
   AxisNuw.Axis[11].Pos14.Reached := FALSE;
   AxisNuw.Axis[11].Pos15.Position := 0.0;
   AxisNuw.Axis[11].Pos15.Speed := 0;
   AxisNuw.Axis[11].Pos15.Reached := FALSE;
   AxisNuw.Axis[11].Pos16.Position := 0.0;
   AxisNuw.Axis[11].Pos16.Speed := 0;
   AxisNuw.Axis[11].Pos16.Reached := FALSE;
   AxisNuw.Axis[11].Pos17.Position := 0.0;
   AxisNuw.Axis[11].Pos17.Speed := 0;
   AxisNuw.Axis[11].Pos17.Reached := FALSE;
   AxisNuw.Axis[11].Pos18.Position := 0.0;
   AxisNuw.Axis[11].Pos18.Speed := 0;
   AxisNuw.Axis[11].Pos18.Reached := FALSE;
   AxisNuw.Axis[11].Pos19.Position := 0.0;
   AxisNuw.Axis[11].Pos19.Speed := 0;
   AxisNuw.Axis[11].Pos19.Reached := FALSE;
   AxisNuw.Axis[11].Pos20.Position := 0.0;
   AxisNuw.Axis[11].Pos20.Speed := 0;
   AxisNuw.Axis[11].Pos20.Reached := FALSE;
   AxisNuw.Axis[11].Pos21.Position := 0.0;
   AxisNuw.Axis[11].Pos21.Speed := 0;
   AxisNuw.Axis[11].Pos21.Reached := FALSE;
   AxisNuw.Axis[11].Pos22.Position := 0.0;
   AxisNuw.Axis[11].Pos22.Speed := 0;
   AxisNuw.Axis[11].Pos22.Reached := FALSE;
   AxisNuw.Axis[11].Pos23.Position := 0.0;
   AxisNuw.Axis[11].Pos23.Speed := 0;
   AxisNuw.Axis[11].Pos23.Reached := FALSE;
   AxisNuw.Axis[11].Pos24.Position := 0.0;
   AxisNuw.Axis[11].Pos24.Speed := 0;
   AxisNuw.Axis[11].Pos24.Reached := FALSE;
   AxisNuw.Axis[11].Pos25.Position := 0.0;
   AxisNuw.Axis[11].Pos25.Speed := 0;
   AxisNuw.Axis[11].Pos25.Reached := FALSE;
   AxisNuw.Axis[11].Pos26.Position := 0.0;
   AxisNuw.Axis[11].Pos26.Speed := 0;
   AxisNuw.Axis[11].Pos26.Reached := FALSE;
   AxisNuw.Axis[11].Pos27.Position := 0.0;
   AxisNuw.Axis[11].Pos27.Speed := 0;
   AxisNuw.Axis[11].Pos27.Reached := FALSE;
   AxisNuw.Axis[11].Pos28.Position := 0.0;
   AxisNuw.Axis[11].Pos28.Speed := 0;
   AxisNuw.Axis[11].Pos28.Reached := FALSE;
   AxisNuw.Axis[11].Pos29.Position := 0.0;
   AxisNuw.Axis[11].Pos29.Speed := 0;
   AxisNuw.Axis[11].Pos29.Reached := FALSE;
   AxisNuw.Axis[11].Pos30.Position := 0.0;
   AxisNuw.Axis[11].Pos30.Speed := 0;
   AxisNuw.Axis[11].Pos30.Reached := FALSE;
   AxisNuw.Axis[12].Pos1.Position := 0.0;
   AxisNuw.Axis[12].Pos1.Speed := 0;
   AxisNuw.Axis[12].Pos1.Reached := FALSE;
   AxisNuw.Axis[12].Pos2.Position := 0.0;
   AxisNuw.Axis[12].Pos2.Speed := 0;
   AxisNuw.Axis[12].Pos2.Reached := FALSE;
   AxisNuw.Axis[12].Pos3.Position := 0.0;
   AxisNuw.Axis[12].Pos3.Speed := 0;
   AxisNuw.Axis[12].Pos3.Reached := FALSE;
   AxisNuw.Axis[12].Pos4.Position := 0.0;
   AxisNuw.Axis[12].Pos4.Speed := 0;
   AxisNuw.Axis[12].Pos4.Reached := FALSE;
   AxisNuw.Axis[12].Pos5.Position := 0.0;
   AxisNuw.Axis[12].Pos5.Speed := 0;
   AxisNuw.Axis[12].Pos5.Reached := FALSE;
   AxisNuw.Axis[12].Pos6.Position := 0.0;
   AxisNuw.Axis[12].Pos6.Speed := 0;
   AxisNuw.Axis[12].Pos6.Reached := FALSE;
   AxisNuw.Axis[12].Pos7.Position := 0.0;
   AxisNuw.Axis[12].Pos7.Speed := 0;
   AxisNuw.Axis[12].Pos7.Reached := FALSE;
   AxisNuw.Axis[12].Pos8.Position := 0.0;
   AxisNuw.Axis[12].Pos8.Speed := 0;
   AxisNuw.Axis[12].Pos8.Reached := FALSE;
   AxisNuw.Axis[12].Pos9.Position := 0.0;
   AxisNuw.Axis[12].Pos9.Speed := 0;
   AxisNuw.Axis[12].Pos9.Reached := FALSE;
   AxisNuw.Axis[12].Pos10.Position := 0.0;
   AxisNuw.Axis[12].Pos10.Speed := 0;
   AxisNuw.Axis[12].Pos10.Reached := FALSE;
   AxisNuw.Axis[12].Pos11.Position := 0.0;
   AxisNuw.Axis[12].Pos11.Speed := 0;
   AxisNuw.Axis[12].Pos11.Reached := FALSE;
   AxisNuw.Axis[12].Pos12.Position := 0.0;
   AxisNuw.Axis[12].Pos12.Speed := 0;
   AxisNuw.Axis[12].Pos12.Reached := FALSE;
   AxisNuw.Axis[12].Pos13.Position := 0.0;
   AxisNuw.Axis[12].Pos13.Speed := 0;
   AxisNuw.Axis[12].Pos13.Reached := FALSE;
   AxisNuw.Axis[12].Pos14.Position := 0.0;
   AxisNuw.Axis[12].Pos14.Speed := 0;
   AxisNuw.Axis[12].Pos14.Reached := FALSE;
   AxisNuw.Axis[12].Pos15.Position := 0.0;
   AxisNuw.Axis[12].Pos15.Speed := 0;
   AxisNuw.Axis[12].Pos15.Reached := FALSE;
   AxisNuw.Axis[12].Pos16.Position := 0.0;
   AxisNuw.Axis[12].Pos16.Speed := 0;
   AxisNuw.Axis[12].Pos16.Reached := FALSE;
   AxisNuw.Axis[12].Pos17.Position := 0.0;
   AxisNuw.Axis[12].Pos17.Speed := 0;
   AxisNuw.Axis[12].Pos17.Reached := FALSE;
   AxisNuw.Axis[12].Pos18.Position := 0.0;
   AxisNuw.Axis[12].Pos18.Speed := 0;
   AxisNuw.Axis[12].Pos18.Reached := FALSE;
   AxisNuw.Axis[12].Pos19.Position := 0.0;
   AxisNuw.Axis[12].Pos19.Speed := 0;
   AxisNuw.Axis[12].Pos19.Reached := FALSE;
   AxisNuw.Axis[12].Pos20.Position := 0.0;
   AxisNuw.Axis[12].Pos20.Speed := 0;
   AxisNuw.Axis[12].Pos20.Reached := FALSE;
   AxisNuw.Axis[12].Pos21.Position := 0.0;
   AxisNuw.Axis[12].Pos21.Speed := 0;
   AxisNuw.Axis[12].Pos21.Reached := FALSE;
   AxisNuw.Axis[12].Pos22.Position := 0.0;
   AxisNuw.Axis[12].Pos22.Speed := 0;
   AxisNuw.Axis[12].Pos22.Reached := FALSE;
   AxisNuw.Axis[12].Pos23.Position := 0.0;
   AxisNuw.Axis[12].Pos23.Speed := 0;
   AxisNuw.Axis[12].Pos23.Reached := FALSE;
   AxisNuw.Axis[12].Pos24.Position := 0.0;
   AxisNuw.Axis[12].Pos24.Speed := 0;
   AxisNuw.Axis[12].Pos24.Reached := FALSE;
   AxisNuw.Axis[12].Pos25.Position := 0.0;
   AxisNuw.Axis[12].Pos25.Speed := 0;
   AxisNuw.Axis[12].Pos25.Reached := FALSE;
   AxisNuw.Axis[12].Pos26.Position := 0.0;
   AxisNuw.Axis[12].Pos26.Speed := 0;
   AxisNuw.Axis[12].Pos26.Reached := FALSE;
   AxisNuw.Axis[12].Pos27.Position := 0.0;
   AxisNuw.Axis[12].Pos27.Speed := 0;
   AxisNuw.Axis[12].Pos27.Reached := FALSE;
   AxisNuw.Axis[12].Pos28.Position := 0.0;
   AxisNuw.Axis[12].Pos28.Speed := 0;
   AxisNuw.Axis[12].Pos28.Reached := FALSE;
   AxisNuw.Axis[12].Pos29.Position := 0.0;
   AxisNuw.Axis[12].Pos29.Speed := 0;
   AxisNuw.Axis[12].Pos29.Reached := FALSE;
   AxisNuw.Axis[12].Pos30.Position := 0.0;
   AxisNuw.Axis[12].Pos30.Speed := 0;
